FUNCTION_BLOCK FB_MY_SQL IMPLEMENTS I_DATABASE
VAR //General
	{attribute 'instance-path'} 
  {attribute 'noinit'} 
	strInstancePath:									                      STRING;
	bInit: 												                          BOOL:=TRUE;
	strFullObjectPath: 								                      STRING;
	stEvent:											                          ST_EVENT;
	bAck:												                            BOOL;
	
END_VAR
VAR   // From FB_init	
	itfLogEvents: 										                      I_HANDLE_EVENTS;
  itfOpMode:											                        I_OP_MODE; 
END_VAR                                      				
VAR	// Step chain control                				
  eSeq, eLastSeq, eNextSeq:					                      E_SEQ_DATABASE; 
                  				
  //eActiveSeqState, eLastActiveSeqState:                 E_SEQ_GENERAL;
	(*
  iInternalSeqStateCase, iLastInternalSeqStateCase:       INT:=0;       
	tonDelay, tonTimeOut, tonStepTime:						          TON;
	tDelay:													                        TIME := T#100MS;
	tTimeOut:												                        TIME := T#100MS;
	tTimeOutExt:											                      TIME := T#100MS;
	bDelayActive, bTimeOutActiveQuit, bTimeOutActiveNoQuit:	BOOL;//Timer Option
	bActiveStep, bDebugAcitve, bDebugNext:					        BOOL;//Debug Option
	i:														                          INT;
 	iError:													                        INT; //ERROR-CODE                    	                   		
	listLastSteps:											                    ARRAY[0..49] OF ST_LAST_STEPS;	
	strExtraInfo:											                      STRING; 
	eStep_Type:												                      E_STEP_STATE_TYPE; 
	bDebugModeActive:										                    BOOL;   
	bWaitForBreakpoint:										                  BOOL;
	bBreakpointActive:										                  BOOL;
	bDebugResume:											                      BOOL;   
	listBreakpoint:											                    ARRAY[0..10] OF  INT;    
*)
i:														                            INT;
stSeqCtrlGeneral:											                    ST_SEQ_CTRL_GEN;     	
END_VAR                                             		
VAR                                                 		
	bMethodeFromExtStarted:									                BOOL;
	bMethodeFromExtActive:									                BOOL;
	bMethodeFromExtDone:									                  BOOL;
	strTemp:												                        STRING;
END_VAR   
VAR
  fbSQLDatabase:            FB_SQLDatabaseEvt(sNetID := '', tTimeout := T#5S);
  fbSQLCommand:             FB_SQLCommandEvt(sNetID := '', tTimeout := T#5S);
  fbPLCDBCmd:               FB_PLCDBCmdEvt(sNetID := '', tTimeout := T#5S);
  fbPLCDBCreateEvt:         FB_PLCDBCreateEvt(sNetID := '', tTimeout := T#5S);
  fbPLCDBReadEvt:           FB_PLCDBReadEvt(sNetID:= '', tTimeout:= T#5S);
  fbPLCDBWriteEvt:          FB_PLCDBWriteEvt(sNetID := '', tTimeout := T#5S);
  udiDBID:                  UDINT;
  pDBID:                    POINTER TO UDINT;
  sCmd:                     STRING(5000);
  sTableName:               T_MaxString;
  sDBSymbolName:            STRING;
  pRecord:                  POINTER TO BYTE;
  cbRecord:                 UDINT;
  pValue:                   POINTER TO BYTE;
  cbValue:                  UDINT;
  pColumnNames:             POINTER TO ARRAY [0..MAX_DBCOLUMNS] OF STRING(50);
  cbColumnNames:            UDINT;
  pTableCfg:                POINTER TO ARRAY[0..MAX_DBCOLUMNS] OF ST_ColumnInfo;
  cbTableCfg:               UDINT;
  sOrderByColumn:           STRING(50);
  eOrderBy:                 E_OrderColumn;
  eOrderType:               E_OrderType;
  nStartIndex:              UDINT;
  nRecordCount:             UDINT;
  pData:                    POINTER TO BYTE;
  pData2:                   POINTER TO ST_StandardRecord;
  cbData:                   UDINT;
  pDatabaseConfig:          POINTER TO BYTE;
  cbDatabaseConfig:         UDINT;
  bCreateXMLConfig:         BOOL;
  sColumnNameToUpdate:      STRING;
  sColumnValToUpdate:       STRING;
  sColumnNameToSet:         STRING;
  sNewVal:                  STRING;
  eDBWriteMode:             E_WriteMode;
  nRingBuffParameter:       UDINT;
  stADSDevice:              ST_ADSDevice;
  stSymbol:                 ST_Symbol;
  pExpression:              POINTER TO BYTE;
  cbExpression:             UDINT;
  pParameter:               POINTER TO ARRAY[0..MAX_DBCOLUMNS] OF ST_ExpParameter;
  cbParameter:              UDINT; 
  pSQLCmd:                  POINTER TO BYTE;
  cbSQLCmd:                 UDINT;
  bResult:                  BOOL;
END_VAR                  	
VAR_TEMP                    	
	iTemp:										INT;
END_VAR

// Set FBs and Interfaces ready after switch internal step
IF stSeqCtrlGeneral.iInternalSeqStateCase <> stSeqCtrlGeneral.iLastInternalSeqStateCase AND NOT stSeqCtrlGeneral.bExitSetReadyState THEN
  IF TRUE
  THEN
    stSeqCtrlGeneral.bExitSetReadyState := TRUE;
  ELSE
    RETURN;
  END_IF
END_IF

stSeqCtrlGeneral.strObject := F_CreateObjectName(strInstancePath);

// First method call
_m_SequenceManager();
//_m_SaveLastStep();

CASE eSeq OF 
  E_SEQ_DATABASE.BASE:;
  
	E_SEQ_DATABASE.INIT: _m_Seq_INIT();
		IF TRUE
		AND (stSeqCtrlGeneral.eActiveSeqState = E_SEQ_GENERAL.DONE) 
		THEN
			eSeq := E_SEQ_DATABASE.BASE;
		END_IF
		
	E_SEQ_DATABASE.SETUP:;
  
	// Process
  E_SEQ_DATABASE.CREATE_DATABASE: _m_Seq_CREATE_DATABASE();
    IF TRUE
		AND (stSeqCtrlGeneral.eActiveSeqState = E_SEQ_GENERAL.DONE) 
		THEN
			eSeq := E_SEQ_DATABASE.BASE;
		END_IF
  
	E_SEQ_DATABASE.CONNECT:         _m_Seq_CONNECT();
    IF TRUE
		AND (stSeqCtrlGeneral.eActiveSeqState = E_SEQ_GENERAL.DONE) 
		THEN
			eSeq := E_SEQ_DATABASE.BASE;
		END_IF
    
  E_SEQ_DATABASE.EXECUTE_SIMPLIFY_CMD:  _m_Seq_EXECUTE_SIMPLIFY_CMD();
    IF TRUE
		AND (stSeqCtrlGeneral.eActiveSeqState = E_SEQ_GENERAL.DONE) 
		THEN
			eSeq := E_SEQ_DATABASE.BASE;
		END_IF
  
  E_SEQ_DATABASE.EXECUTE_CMD:     _m_Seq_EXECUTE_CMD();
    IF TRUE
		AND (stSeqCtrlGeneral.eActiveSeqState = E_SEQ_GENERAL.DONE) 
		THEN
			eSeq := E_SEQ_DATABASE.BASE;
		END_IF
    
  E_SEQ_DATABASE.TABLE_EXIST_CHECK:     _m_Seq_TABLE_EXIST_CHECK();
    IF TRUE
		AND (stSeqCtrlGeneral.eActiveSeqState = E_SEQ_GENERAL.DONE) 
		THEN
			eSeq := E_SEQ_DATABASE.BASE;
		END_IF
  
  E_SEQ_DATABASE.CREATE_TABLE:    _m_Seq_CREATE_TABLE();
    IF TRUE
		AND (stSeqCtrlGeneral.eActiveSeqState = E_SEQ_GENERAL.DONE) 
		THEN
			eSeq := E_SEQ_DATABASE.BASE;
		END_IF
  
  E_SEQ_DATABASE.WRITE:           _m_Seq_WRITE();
    IF TRUE
		AND (stSeqCtrlGeneral.eActiveSeqState = E_SEQ_GENERAL.DONE) 
		THEN
			eSeq := E_SEQ_DATABASE.BASE;
		END_IF
  
  E_SEQ_DATABASE.WRITE_STRUCT:    _m_Seq_WRITE_STRUCT();
    IF TRUE
		AND (stSeqCtrlGeneral.eActiveSeqState = E_SEQ_GENERAL.DONE) 
		THEN
			eSeq := E_SEQ_DATABASE.BASE;
		END_IF
  
  E_SEQ_DATABASE.WRITE_BY_SYMBOL: _m_Seq_WRITE_BY_SYMBOL();
    IF TRUE
		AND (stSeqCtrlGeneral.eActiveSeqState = E_SEQ_GENERAL.DONE) 
		THEN
			eSeq := E_SEQ_DATABASE.BASE;
		END_IF
  
  E_SEQ_DATABASE.OVERWRITE:       _m_Seq_OVERWRITE();
    IF TRUE
		AND (stSeqCtrlGeneral.eActiveSeqState = E_SEQ_GENERAL.DONE) 
		THEN
			eSeq := E_SEQ_DATABASE.BASE;
		END_IF
  
  E_SEQ_DATABASE.READ:            _m_Seq_READ();
    IF TRUE
		AND (stSeqCtrlGeneral.eActiveSeqState = E_SEQ_GENERAL.DONE) 
		THEN
			eSeq := E_SEQ_DATABASE.BASE;
		END_IF
  
  E_SEQ_DATABASE.READ_STRUCT:     _m_Seq_READ_STRUCT();
    IF TRUE
		AND (stSeqCtrlGeneral.eActiveSeqState = E_SEQ_GENERAL.DONE) 
		THEN
			eSeq := E_SEQ_DATABASE.BASE;
		END_IF
  
  E_SEQ_DATABASE.CLEAR_TABLE:     _m_Seq_CLEAR_TABLE();
    IF TRUE
		AND (stSeqCtrlGeneral.eActiveSeqState = E_SEQ_GENERAL.DONE) 
		THEN
			eSeq := E_SEQ_DATABASE.BASE;
		END_IF
  
  E_SEQ_DATABASE.DELETE_TABLE:    _m_Seq_DELETE_TABLE();
    IF TRUE
		AND (stSeqCtrlGeneral.eActiveSeqState = E_SEQ_GENERAL.DONE) 
		THEN
			eSeq := E_SEQ_DATABASE.BASE;
		END_IF
  
  E_SEQ_DATABASE.DISCONNECT:      _m_Seq_DISCONNECT();
    IF TRUE
		AND (stSeqCtrlGeneral.eActiveSeqState = E_SEQ_GENERAL.DONE) 
		THEN
			eSeq := E_SEQ_DATABASE.BASE;
		END_IF

  // End
	E_SEQ_DATABASE.END:;
	E_SEQ_DATABASE.ERROR_SEQ:;	
END_CASE

strTemp:=TO_STRING(eSeq);

METHOD PRIVATE _m_DebugManager
VAR_INPUT
	iStepID: int;
END_VAR
IF TRUE
AND THIS^.stSeqCtrlGeneral.bDebugModeActive 
AND NOT THIS^.stSeqCtrlGeneral.bActiveStep
THEN


THIS^.stSeqCtrlGeneral.bBreakpointActive:=FALSE;

FOR i:=0 TO 10 DO
	
	IF TRUE
	AND iStepID=THIS^.stSeqCtrlGeneral.listBreakpoint[i] 
	AND iStepID<>0
	THEN
		EXIT;
	END_IF
END_FOR
IF (i<=10) THEN
	THIS^.stSeqCtrlGeneral.bBreakpointActive:=TRUE;
END_IF

END_IF
END_METHOD

METHOD PRIVATE _m_Delay : BOOL
VAR_INPUT
	DelayTime:	TIME;
END_VAR
THIS^.stSeqCtrlGeneral.bDelayActive:=TRUE;
THIS^.stSeqCtrlGeneral.tDelay:=DelayTime;
_m_Delay:=FALSE;
IF THIS^.stSeqCtrlGeneral.tonDelay.Q THEN
	_m_Delay:=TRUE;
END_IF
END_METHOD

METHOD PRIVATE _m_GeneralStepSetting : BOOL
VAR_INPUT
	StepType:			    	E_STEP_STATE_TYPE;
	InfoTextID:					STRING(20);
	EnableDebug:	   			BOOL;	
	
END_VAR
IF THIS^.stSeqCtrlGeneral.bActiveStep THEN
	THIS^.stSeqCtrlGeneral.eStep_Type:=StepType;
	THIS^.stSeqCtrlGeneral.strExtraInfo:= GenLib.F_RET_TXTLIST_ENTRY(strPortNr:='851',strID:='',strTxtLstName:=InfoTextID);
END_IF
END_METHOD

METHOD PRIVATE _m_SaveLastStep : BOOL
VAR_INPUT
END_VAR
VAR
	i: dint;
END_VAR
IF NOT THIS^.stSeqCtrlGeneral.bActiveStep THEN
	
	FOR i:=49 TO 1 BY -1 DO
			stSeqCtrlGeneral.listLastSteps[i].strStepName:=stSeqCtrlGeneral.listLastSteps[i-1].strStepName;
			stSeqCtrlGeneral.listLastSteps[i].tStepTime:=stSeqCtrlGeneral.listLastSteps[i-1].tStepTime;
			stSeqCtrlGeneral.listLastSteps[i].tDelayTime:=stSeqCtrlGeneral.listLastSteps[i-1].tDelayTime;
	END_FOR
	stSeqCtrlGeneral.listLastSteps[0].strStepName:=TO_STRING(THIS^.eSeq);
	stSeqCtrlGeneral.listLastSteps[1].tStepTime:=THIS^.stSeqCtrlGeneral.tonStepTime.ET;
	stSeqCtrlGeneral.listLastSteps[1].tStepTime:=THIS^.stSeqCtrlGeneral.tonDelay.ET;
ELSE
	stSeqCtrlGeneral.listLastSteps[0].tStepTime:=THIS^.stSeqCtrlGeneral.tonStepTime.ET;
	stSeqCtrlGeneral.listLastSteps[0].tDelayTime:=THIS^.stSeqCtrlGeneral.tonDelay.ET;	
END_IF
END_METHOD

METHOD PRIVATE _m_Seq_CLEAR_TABLE : E_SEQ_PROCESS
VAR_INPUT
END_VAR
VAR
	ActiveSeq: STRING;
END_VAR
VAR
	
END_VAR
//THIS^._m_GeneralStepSetting(StepType:=E_STEP_STATE_TYPE.INIT,
ActiveSeq := TO_STRING(THIS^.eSeq);

CASE THIS^.stSeqCtrlGeneral.eActiveSeqState OF
E_SEQ_GENERAL.READY:;

	
E_SEQ_GENERAL.EXECUTE:;
	IF TRUE
	THEN
		THIS^.stSeqCtrlGeneral.eActiveSeqState := E_SEQ_GENERAL.RESET;
	END_IF
  
E_SEQ_GENERAL.RESET:;
	stSeqCtrlGeneral.iInternalSeqStateCase := 0;
	IF TRUE
	THEN
		THIS^.stSeqCtrlGeneral.eActiveSeqState := E_SEQ_GENERAL.BUSY;
	END_IF
  
E_SEQ_GENERAL.BUSY:;
	CASE THIS^.stSeqCtrlGeneral.iInternalSeqStateCase OF
    0:  // Connect to database
      IF TRUE 
      AND NOT THIS^.fbSQLDatabase.bConnected
			THEN 
        IF THIS^.fbSQLDatabase.Connect(THIS^.udiDBID) THEN
          IF THIS^.fbSQLDatabase.bError THEN
            THIS^.stSeqCtrlGeneral.eActiveSeqState := E_SEQ_GENERAL.ERROR;
          ELSE
            THIS^.stSeqCtrlGeneral.iInternalSeqStateCase := 10;
          END_IF
        END_IF
      ELSE
        THIS^.stSeqCtrlGeneral.iInternalSeqStateCase := 10;
			END_IF
      
		10:	// Create command
      IF TRUE 
			THEN 
        sCmd := 'DELETE FROM `';
        sCmd := CONCAT(sCmd, sTableName);
        sCmd := CONCAT(sCmd, '`');
        IF fbSQLDatabase.CreateCmd(ADR(fbSQLCommand)) THEN
          IF fbSqlDatabase.bError THEN
            THIS^.stSeqCtrlGeneral.eActiveSeqState := E_SEQ_GENERAL.ERROR;
          ELSE
            THIS^.stSeqCtrlGeneral.iInternalSeqStateCase := 20;  
          END_IF
        END_IF
			END_IF
      
		20: // Execute command
      IF TRUE 
			THEN
        IF fbSQLCommand.Execute(ADR(sCmd), SIZEOF(sCmd)) THEN
          IF fbSQLCommand.bError THEN
            THIS^.stSeqCtrlGeneral.eActiveSeqState := E_SEQ_GENERAL.ERROR;
          ELSE
            THIS^.stSeqCtrlGeneral.iInternalSeqStateCase := 30;
          END_IF
	      END_IF
			END_IF
      
    30:	// Disconnect
      IF TRUE 
			THEN 
        IF fbSQLDatabase.Disconnect() THEN
          IF fbSqlDatabase.bError THEN
            THIS^.stSeqCtrlGeneral.eActiveSeqState := E_SEQ_GENERAL.ERROR;
          ELSE
            THIS^.stSeqCtrlGeneral.iInternalSeqStateCase := 1000;
          END_IF
        END_IF
			END_IF
      
	ELSE
		THIS^.stSeqCtrlGeneral.eActiveSeqState := E_SEQ_GENERAL.DONE;  
	END_CASE
	THIS^.stSeqCtrlGeneral.strExtraInfo := CONCAT('Internal state: ', TO_STRING(THIS^.stSeqCtrlGeneral.iInternalSeqStateCase));

E_SEQ_GENERAL.DONE:;

E_SEQ_GENERAL.ERROR:;

E_SEQ_GENERAL.TIME_OUT:; 
IF TRUE
AND THIS^.stSeqCtrlGeneral.bTimeOutActiveQuit 
THEN
  THIS^.stSeqCtrlGeneral.strExtraInfo := 'Bitte quittieren und erneut testen';
  IF TRUE
  //AND itfOpMode.P_QUIT
  THEN
    THIS^.stSeqCtrlGeneral.eActiveSeqState := E_SEQ_GENERAL.EXECUTE;
	END_IF
  
END_IF

ELSE
  THIS^.stSeqCtrlGeneral.eActiveSeqState := E_SEQ_GENERAL.ERROR;
END_CASE
END_METHOD

METHOD PRIVATE _m_Seq_CONNECT : E_SEQ_PROCESS
VAR_INPUT
END_VAR
VAR
	ActiveSeq: STRING;
END_VAR
VAR
	
END_VAR
//THIS^._m_GeneralStepSetting(StepType:=E_STEP_STATE_TYPE.INIT,
ActiveSeq := TO_STRING(THIS^.eSeq);

CASE THIS^.stSeqCtrlGeneral.eActiveSeqState OF
E_SEQ_GENERAL.READY:;

	
E_SEQ_GENERAL.EXECUTE:;
	IF TRUE
	THEN
		THIS^.stSeqCtrlGeneral.eActiveSeqState := E_SEQ_GENERAL.RESET;
	END_IF
  
E_SEQ_GENERAL.RESET:;
	stSeqCtrlGeneral.iInternalSeqStateCase := 0;
	IF TRUE
	THEN
		THIS^.stSeqCtrlGeneral.eActiveSeqState := E_SEQ_GENERAL.BUSY;
	END_IF
  
E_SEQ_GENERAL.BUSY:;
	CASE THIS^.stSeqCtrlGeneral.iInternalSeqStateCase OF
		0:	// Entrance step --> Connect
      IF TRUE 
      AND NOT THIS^.fbSQLDatabase.bConnected
			THEN 
        IF THIS^.fbSQLDatabase.Connect(THIS^.udiDBID) THEN
          IF THIS^.fbSQLDatabase.bError THEN
            THIS^.stSeqCtrlGeneral.eActiveSeqState := E_SEQ_GENERAL.ERROR;
          ELSE
            THIS^.stSeqCtrlGeneral.iInternalSeqStateCase := 1000;
          END_IF
        END_IF
      ELSE
        THIS^.stSeqCtrlGeneral.iInternalSeqStateCase := 1000;
			END_IF
      
	ELSE
		THIS^.stSeqCtrlGeneral.eActiveSeqState := E_SEQ_GENERAL.DONE;  
	END_CASE
	THIS^.stSeqCtrlGeneral.strExtraInfo := CONCAT('Internal state: ', TO_STRING(THIS^.stSeqCtrlGeneral.iInternalSeqStateCase));

E_SEQ_GENERAL.DONE:;

E_SEQ_GENERAL.ERROR:;

E_SEQ_GENERAL.TIME_OUT:; 
IF TRUE
AND THIS^.stSeqCtrlGeneral.bTimeOutActiveQuit 
THEN
  THIS^.stSeqCtrlGeneral.strExtraInfo := 'Bitte quittieren und erneut testen';
  IF TRUE
  //AND itfOpMode.P_QUIT
  THEN
    THIS^.stSeqCtrlGeneral.eActiveSeqState := E_SEQ_GENERAL.EXECUTE;
	END_IF
  
END_IF

ELSE
  THIS^.stSeqCtrlGeneral.eActiveSeqState := E_SEQ_GENERAL.ERROR;
END_CASE
END_METHOD

METHOD PRIVATE _m_Seq_CREATE_DATABASE : E_SEQ_PROCESS
VAR_INPUT
END_VAR
VAR
	ActiveSeq: STRING;
END_VAR
VAR
  stTemp:                     STRING;
END_VAR
//THIS^._m_GeneralStepSetting(StepType:=E_STEP_STATE_TYPE.INIT,
ActiveSeq := TO_STRING(THIS^.eSeq);

CASE THIS^.stSeqCtrlGeneral.eActiveSeqState OF
E_SEQ_GENERAL.READY:;

	
E_SEQ_GENERAL.EXECUTE:;
	IF TRUE
	THEN
		THIS^.stSeqCtrlGeneral.eActiveSeqState := E_SEQ_GENERAL.RESET;
	END_IF
  
E_SEQ_GENERAL.RESET:;
	stSeqCtrlGeneral.iInternalSeqStateCase := 0;
	IF TRUE
	THEN
		THIS^.stSeqCtrlGeneral.eActiveSeqState := E_SEQ_GENERAL.BUSY;
	END_IF
  
E_SEQ_GENERAL.BUSY:;
	CASE THIS^.stSeqCtrlGeneral.iInternalSeqStateCase OF
    0:	// Create database
      IF TRUE 
			THEN
        IF fbPLCDBCreateEvt.Database(
          pDatabaseConfig:= pDatabaseConfig,
          cbDatabaseConfig:= cbDatabaseConfig,
          bCreateXMLConfig:= bCreateXMLConfig,
          pDBID := pDBID)
        THEN
          IF fbPLCDBCreateEvt.bError THEN
            THIS^.stSeqCtrlGeneral.eActiveSeqState := E_SEQ_GENERAL.ERROR; 
          ELSE
            THIS^.stSeqCtrlGeneral.iInternalSeqStateCase := 1000;
          END_IF
        END_IF
      END_IF
      
	ELSE
		THIS^.stSeqCtrlGeneral.eActiveSeqState := E_SEQ_GENERAL.DONE;  
	END_CASE
	THIS^.stSeqCtrlGeneral.strExtraInfo := CONCAT('Internal state: ', TO_STRING(THIS^.stSeqCtrlGeneral.iInternalSeqStateCase));

E_SEQ_GENERAL.DONE:;

E_SEQ_GENERAL.ERROR:;

E_SEQ_GENERAL.TIME_OUT:; 
IF TRUE
AND THIS^.stSeqCtrlGeneral.bTimeOutActiveQuit 
THEN
  THIS^.stSeqCtrlGeneral.strExtraInfo := 'Bitte quittieren und erneut testen';
  IF TRUE
  //AND itfOpMode.P_QUIT
  THEN
    THIS^.stSeqCtrlGeneral.eActiveSeqState := E_SEQ_GENERAL.EXECUTE;
	END_IF
  
END_IF

ELSE
  THIS^.stSeqCtrlGeneral.eActiveSeqState := E_SEQ_GENERAL.ERROR;
END_CASE
END_METHOD

METHOD PRIVATE _m_Seq_CREATE_TABLE : E_SEQ_PROCESS
VAR_INPUT
END_VAR
VAR
	ActiveSeq: STRING;
END_VAR
VAR
  stTemp:                     STRING;
END_VAR
//THIS^._m_GeneralStepSetting(StepType:=E_STEP_STATE_TYPE.INIT,
ActiveSeq := TO_STRING(THIS^.eSeq);

CASE THIS^.stSeqCtrlGeneral.eActiveSeqState OF
E_SEQ_GENERAL.READY:;

	
E_SEQ_GENERAL.EXECUTE:;
	IF TRUE
	THEN
		THIS^.stSeqCtrlGeneral.eActiveSeqState := E_SEQ_GENERAL.RESET;
	END_IF
  
E_SEQ_GENERAL.RESET:;
	stSeqCtrlGeneral.iInternalSeqStateCase := 0;
	IF TRUE
	THEN
		THIS^.stSeqCtrlGeneral.eActiveSeqState := E_SEQ_GENERAL.BUSY;
	END_IF
  
E_SEQ_GENERAL.BUSY:;
	CASE THIS^.stSeqCtrlGeneral.iInternalSeqStateCase OF
    0:	// Create table
      IF TRUE 
			THEN
        IF fbPLCDBCreateEvt.Table(hDBID:= udiDBID,
                                  sTableName:= sTableName, 
                                  pTableCfg:= THIS^.pTableCfg, 
                                  cbTableCfg:= THIS^.cbTableCfg)
        THEN
          IF fbPLCDBCreateEvt.bError THEN
            THIS^.stSeqCtrlGeneral.eActiveSeqState := E_SEQ_GENERAL.ERROR; 
          ELSE
            THIS^.stSeqCtrlGeneral.iInternalSeqStateCase := 1000;
          END_IF
        END_IF
      END_IF
      
	ELSE
		THIS^.stSeqCtrlGeneral.eActiveSeqState := E_SEQ_GENERAL.DONE;  
	END_CASE
	THIS^.stSeqCtrlGeneral.strExtraInfo := CONCAT('Internal state: ', TO_STRING(THIS^.stSeqCtrlGeneral.iInternalSeqStateCase));

E_SEQ_GENERAL.DONE:;

E_SEQ_GENERAL.ERROR:;

E_SEQ_GENERAL.TIME_OUT:; 
IF TRUE
AND THIS^.stSeqCtrlGeneral.bTimeOutActiveQuit 
THEN
  THIS^.stSeqCtrlGeneral.strExtraInfo := 'Bitte quittieren und erneut testen';
  IF TRUE
  //AND itfOpMode.P_QUIT
  THEN
    THIS^.stSeqCtrlGeneral.eActiveSeqState := E_SEQ_GENERAL.EXECUTE;
	END_IF
  
END_IF

ELSE
  THIS^.stSeqCtrlGeneral.eActiveSeqState := E_SEQ_GENERAL.ERROR;
END_CASE
END_METHOD

METHOD PRIVATE _m_Seq_DELETE_TABLE : E_SEQ_PROCESS
VAR_INPUT
END_VAR
VAR
	ActiveSeq: STRING;
END_VAR
VAR
	
END_VAR
//THIS^._m_GeneralStepSetting(StepType:=E_STEP_STATE_TYPE.INIT,
ActiveSeq := TO_STRING(THIS^.eSeq);

CASE THIS^.stSeqCtrlGeneral.eActiveSeqState OF
E_SEQ_GENERAL.READY:;

	
E_SEQ_GENERAL.EXECUTE:;
	IF TRUE
	THEN
		THIS^.stSeqCtrlGeneral.eActiveSeqState := E_SEQ_GENERAL.RESET;
	END_IF
  
E_SEQ_GENERAL.RESET:;
	stSeqCtrlGeneral.iInternalSeqStateCase := 0;
	IF TRUE
	THEN
		THIS^.stSeqCtrlGeneral.eActiveSeqState := E_SEQ_GENERAL.BUSY;
	END_IF
  
E_SEQ_GENERAL.BUSY:;
	CASE THIS^.stSeqCtrlGeneral.iInternalSeqStateCase OF
    0:  // Connect to database
      IF TRUE 
      AND NOT THIS^.fbSQLDatabase.bConnected
			THEN 
        IF THIS^.fbSQLDatabase.Connect(THIS^.udiDBID) THEN
          IF THIS^.fbSQLDatabase.bError THEN
            THIS^.stSeqCtrlGeneral.eActiveSeqState := E_SEQ_GENERAL.ERROR;
          ELSE
            THIS^.stSeqCtrlGeneral.iInternalSeqStateCase := 10;
          END_IF
        END_IF
      ELSE
        THIS^.stSeqCtrlGeneral.iInternalSeqStateCase := 10;
			END_IF
      
		10:	// Create command
      IF TRUE 
			THEN 
        sCmd := 'DROP TABLE `';
        sCmd := CONCAT(sCmd, sTableName);
        sCmd := CONCAT(sCmd, '`');
        IF fbSQLDatabase.CreateCmd(ADR(fbSQLCommand)) THEN
          IF fbSqlDatabase.bError THEN
            THIS^.stSeqCtrlGeneral.eActiveSeqState := E_SEQ_GENERAL.ERROR;
          ELSE
            THIS^.stSeqCtrlGeneral.iInternalSeqStateCase := 20;  
          END_IF
        END_IF
			END_IF
      
		20: // Execute command
      IF TRUE 
			THEN
        IF fbSQLCommand.Execute(ADR(sCmd), SIZEOF(sCmd)) THEN
          IF fbSQLCommand.bError THEN
            THIS^.stSeqCtrlGeneral.eActiveSeqState := E_SEQ_GENERAL.ERROR;
          ELSE
            THIS^.stSeqCtrlGeneral.iInternalSeqStateCase := 30;
          END_IF
	      END_IF
			END_IF
      
    30:	// Disconnect
      IF TRUE 
			THEN 
        IF fbSQLDatabase.Disconnect() THEN
          IF fbSqlDatabase.bError THEN
            THIS^.stSeqCtrlGeneral.eActiveSeqState := E_SEQ_GENERAL.ERROR;
          ELSE
            THIS^.stSeqCtrlGeneral.iInternalSeqStateCase := 1000;
          END_IF
        END_IF
			END_IF
      
	ELSE
		THIS^.stSeqCtrlGeneral.eActiveSeqState := E_SEQ_GENERAL.DONE;  
	END_CASE
	THIS^.stSeqCtrlGeneral.strExtraInfo := CONCAT('Internal state: ', TO_STRING(THIS^.stSeqCtrlGeneral.iInternalSeqStateCase));

E_SEQ_GENERAL.DONE:;

E_SEQ_GENERAL.ERROR:;

E_SEQ_GENERAL.TIME_OUT:; 
IF TRUE
AND THIS^.stSeqCtrlGeneral.bTimeOutActiveQuit 
THEN
  THIS^.stSeqCtrlGeneral.strExtraInfo := 'Bitte quittieren und erneut testen';
  IF TRUE
  //AND itfOpMode.P_QUIT
  THEN
    THIS^.stSeqCtrlGeneral.eActiveSeqState := E_SEQ_GENERAL.EXECUTE;
	END_IF
  
END_IF

ELSE
  THIS^.stSeqCtrlGeneral.eActiveSeqState := E_SEQ_GENERAL.ERROR;
END_CASE
END_METHOD

METHOD PRIVATE _m_Seq_DISCONNECT : E_SEQ_PROCESS
VAR_INPUT
END_VAR
VAR
	ActiveSeq: STRING;
END_VAR
VAR
	
END_VAR
//THIS^._m_GeneralStepSetting(StepType:=E_STEP_STATE_TYPE.INIT,
ActiveSeq := TO_STRING(THIS^.eSeq);

CASE THIS^.stSeqCtrlGeneral.eActiveSeqState OF
E_SEQ_GENERAL.READY:;

	
E_SEQ_GENERAL.EXECUTE:;
	IF TRUE
	THEN
		THIS^.stSeqCtrlGeneral.eActiveSeqState := E_SEQ_GENERAL.RESET;
	END_IF
  
E_SEQ_GENERAL.RESET:;
	stSeqCtrlGeneral.iInternalSeqStateCase := 0;
	IF TRUE
	THEN
		THIS^.stSeqCtrlGeneral.eActiveSeqState := E_SEQ_GENERAL.BUSY;
	END_IF
  
E_SEQ_GENERAL.BUSY:;
	CASE THIS^.stSeqCtrlGeneral.iInternalSeqStateCase OF
		0:	// Entrance step --> Disconnect
      IF TRUE 
			THEN 
        IF fbSQLDatabase.Disconnect() THEN
          IF fbSqlDatabase.bError THEN
            THIS^.stSeqCtrlGeneral.eActiveSeqState := E_SEQ_GENERAL.ERROR;
          ELSE
            THIS^.stSeqCtrlGeneral.iInternalSeqStateCase := 1000;
          END_IF
        END_IF
			END_IF
      
	ELSE
		THIS^.stSeqCtrlGeneral.eActiveSeqState := E_SEQ_GENERAL.DONE;  
	END_CASE
	THIS^.stSeqCtrlGeneral.strExtraInfo := CONCAT('Internal state: ', TO_STRING(THIS^.stSeqCtrlGeneral.iInternalSeqStateCase));

E_SEQ_GENERAL.DONE:;

E_SEQ_GENERAL.ERROR:;

E_SEQ_GENERAL.TIME_OUT:; 
IF TRUE
AND THIS^.stSeqCtrlGeneral.bTimeOutActiveQuit 
THEN
  THIS^.stSeqCtrlGeneral.strExtraInfo := 'Bitte quittieren und erneut testen';
  IF TRUE
  //AND itfOpMode.P_QUIT
  THEN
    THIS^.stSeqCtrlGeneral.eActiveSeqState := E_SEQ_GENERAL.EXECUTE;
	END_IF
  
END_IF

ELSE
  THIS^.stSeqCtrlGeneral.eActiveSeqState := E_SEQ_GENERAL.ERROR;
END_CASE
END_METHOD

METHOD PRIVATE _m_Seq_EXECUTE_CMD : E_SEQ_PROCESS
VAR_INPUT
END_VAR
VAR
	ActiveSeq: STRING;
END_VAR
//THIS^._m_GeneralStepSetting(StepType:=E_STEP_STATE_TYPE.INIT,
ActiveSeq := TO_STRING(THIS^.eSeq);

CASE THIS^.stSeqCtrlGeneral.eActiveSeqState OF
E_SEQ_GENERAL.READY:;

	
E_SEQ_GENERAL.EXECUTE:;
	IF TRUE
	THEN
		THIS^.stSeqCtrlGeneral.eActiveSeqState := E_SEQ_GENERAL.RESET;
	END_IF
  
E_SEQ_GENERAL.RESET:;
	stSeqCtrlGeneral.iInternalSeqStateCase := 0;
	IF TRUE
	THEN
		THIS^.stSeqCtrlGeneral.eActiveSeqState := E_SEQ_GENERAL.BUSY;
	END_IF
  
E_SEQ_GENERAL.BUSY:;
	CASE THIS^.stSeqCtrlGeneral.iInternalSeqStateCase OF
    0:	// Execute command
      IF TRUE 
			THEN 
        IF fbPLCDBCmd.Execute(hDBID:= THIS^.udiDBID, 
                              pExpression:= pExpression, 
                              cbExpression:= cbExpression, 
                              pData:= pData, 
                              cbData:= cbData, 
                              pParameter:= pParameter, 
                              cbParameter:= cbParameter) 
        THEN
          IF fbPLCDBWriteEvt.bError THEN
            THIS^.stSeqCtrlGeneral.eActiveSeqState := E_SEQ_GENERAL.ERROR; 
          ELSE
            THIS^.stSeqCtrlGeneral.iInternalSeqStateCase := 1000;
          END_IF
        END_IF
			END_IF
      
	ELSE
		THIS^.stSeqCtrlGeneral.eActiveSeqState := E_SEQ_GENERAL.DONE;  
	END_CASE
	THIS^.stSeqCtrlGeneral.strExtraInfo := CONCAT('Internal state: ', TO_STRING(THIS^.stSeqCtrlGeneral.iInternalSeqStateCase));

E_SEQ_GENERAL.DONE:;

E_SEQ_GENERAL.ERROR:;

E_SEQ_GENERAL.TIME_OUT:; 
IF TRUE
AND THIS^.stSeqCtrlGeneral.bTimeOutActiveQuit 
THEN
  THIS^.stSeqCtrlGeneral.strExtraInfo := 'Bitte quittieren und erneut testen';
  IF TRUE
  //AND itfOpMode.P_QUIT
  THEN
    THIS^.stSeqCtrlGeneral.eActiveSeqState := E_SEQ_GENERAL.EXECUTE;
	END_IF
  
END_IF

ELSE
  THIS^.stSeqCtrlGeneral.eActiveSeqState := E_SEQ_GENERAL.ERROR;
END_CASE
END_METHOD

METHOD PRIVATE _m_Seq_EXECUTE_SIMPLIFY_CMD : E_SEQ_PROCESS
VAR_INPUT
END_VAR
VAR
	ActiveSeq: STRING;
END_VAR
//THIS^._m_GeneralStepSetting(StepType:=E_STEP_STATE_TYPE.INIT,
ActiveSeq := TO_STRING(THIS^.eSeq);

CASE THIS^.stSeqCtrlGeneral.eActiveSeqState OF
E_SEQ_GENERAL.READY:;

	
E_SEQ_GENERAL.EXECUTE:;
	IF TRUE
	THEN
		THIS^.stSeqCtrlGeneral.eActiveSeqState := E_SEQ_GENERAL.RESET;
	END_IF
  
E_SEQ_GENERAL.RESET:;
	stSeqCtrlGeneral.iInternalSeqStateCase := 0;
	IF TRUE
	THEN
		THIS^.stSeqCtrlGeneral.eActiveSeqState := E_SEQ_GENERAL.BUSY;
	END_IF
  
E_SEQ_GENERAL.BUSY:;
	CASE THIS^.stSeqCtrlGeneral.iInternalSeqStateCase OF
    0:  // Connect to database
      IF TRUE 
      AND NOT THIS^.fbSQLDatabase.bConnected
			THEN 
        IF THIS^.fbSQLDatabase.Connect(THIS^.udiDBID) THEN
          IF THIS^.fbSQLDatabase.bError THEN
            THIS^.stSeqCtrlGeneral.eActiveSeqState := E_SEQ_GENERAL.ERROR;
          ELSE
            THIS^.stSeqCtrlGeneral.iInternalSeqStateCase := 10;
          END_IF
        END_IF
      ELSE
        THIS^.stSeqCtrlGeneral.iInternalSeqStateCase := 10;
			END_IF

    10:	// Execute command
      IF TRUE 
			THEN 
        IF fbSQLCommand.Execute(THIS^.pSQLCmd, THIS^.cbSQLCmd) THEN
          IF fbPLCDBWriteEvt.bError THEN
            THIS^.stSeqCtrlGeneral.eActiveSeqState := E_SEQ_GENERAL.ERROR; 
          ELSE
            THIS^.stSeqCtrlGeneral.iInternalSeqStateCase := 20;
          END_IF
        END_IF
			END_IF
      
    20:	// Disconnect
      IF TRUE 
			THEN 
        IF fbSQLDatabase.Disconnect() THEN
          IF fbSqlDatabase.bError THEN
            THIS^.stSeqCtrlGeneral.eActiveSeqState := E_SEQ_GENERAL.ERROR;
          ELSE
            THIS^.stSeqCtrlGeneral.iInternalSeqStateCase := 1000;
          END_IF
        END_IF
			END_IF
      
	ELSE
		THIS^.stSeqCtrlGeneral.eActiveSeqState := E_SEQ_GENERAL.DONE;  
	END_CASE
	THIS^.stSeqCtrlGeneral.strExtraInfo := CONCAT('Internal state: ', TO_STRING(THIS^.stSeqCtrlGeneral.iInternalSeqStateCase));

E_SEQ_GENERAL.DONE:;

E_SEQ_GENERAL.ERROR:;

E_SEQ_GENERAL.TIME_OUT:; 
IF TRUE
AND THIS^.stSeqCtrlGeneral.bTimeOutActiveQuit 
THEN
  THIS^.stSeqCtrlGeneral.strExtraInfo := 'Bitte quittieren und erneut testen';
  IF TRUE
  //AND itfOpMode.P_QUIT
  THEN
    THIS^.stSeqCtrlGeneral.eActiveSeqState := E_SEQ_GENERAL.EXECUTE;
	END_IF
  
END_IF

ELSE
  THIS^.stSeqCtrlGeneral.eActiveSeqState := E_SEQ_GENERAL.ERROR;
END_CASE
END_METHOD

METHOD PRIVATE _m_Seq_INIT : E_SEQ_PROCESS
VAR_INPUT
END_VAR
VAR
	ActiveSeq: STRING;
END_VAR
VAR
	
END_VAR
//THIS^._m_GeneralStepSetting(StepType:=E_STEP_STATE_TYPE.INIT,
ActiveSeq := TO_STRING(THIS^.eSeq);

CASE THIS^.stSeqCtrlGeneral.eActiveSeqState OF
E_SEQ_GENERAL.READY:;

	
E_SEQ_GENERAL.EXECUTE:;
	IF TRUE
	THEN
		THIS^.stSeqCtrlGeneral.eActiveSeqState := E_SEQ_GENERAL.RESET;
	END_IF
E_SEQ_GENERAL.RESET:;
	stSeqCtrlGeneral.iInternalSeqStateCase := 0;
  
	IF TRUE
	THEN
		THIS^.stSeqCtrlGeneral.eActiveSeqState := E_SEQ_GENERAL.BUSY;
	END_IF
E_SEQ_GENERAL.BUSY:;
	CASE THIS^.stSeqCtrlGeneral.iInternalSeqStateCase OF
		0:	// Entrance step
      IF TRUE
			THEN 
				IF fbSQLDatabase.Disconnect() THEN
          IF fbSqlDatabase.bError THEN
            THIS^.stSeqCtrlGeneral.eActiveSeqState := E_SEQ_GENERAL.ERROR;
          ELSE
            THIS^.stSeqCtrlGeneral.iInternalSeqStateCase := 1000;
          END_IF
        END_IF
			END_IF
      
	ELSE
		THIS^.stSeqCtrlGeneral.eActiveSeqState := E_SEQ_GENERAL.DONE;  
	END_CASE
	THIS^.stSeqCtrlGeneral.strExtraInfo := CONCAT('Internal state: ', TO_STRING(THIS^.stSeqCtrlGeneral.iInternalSeqStateCase));
E_SEQ_GENERAL.DONE:;
E_SEQ_GENERAL.ERROR:;
E_SEQ_GENERAL.TIME_OUT:; 

IF TRUE
AND THIS^.stSeqCtrlGeneral.bTimeOutActiveQuit 
THEN
  THIS^.stSeqCtrlGeneral.strExtraInfo := 'Bitte quittieren und erneut testen';
  IF TRUE
  //AND itfOpMode.P_QUIT
  THEN
    THIS^.stSeqCtrlGeneral.eActiveSeqState := E_SEQ_GENERAL.EXECUTE;
	END_IF
  
END_IF

ELSE
  THIS^.stSeqCtrlGeneral.eActiveSeqState := E_SEQ_GENERAL.ERROR;
END_CASE
END_METHOD

METHOD PRIVATE _m_Seq_OVERWRITE : E_SEQ_PROCESS
VAR_INPUT
END_VAR
VAR
	ActiveSeq: STRING;
END_VAR
VAR
	sTableName:                 STRING;
  sColumnNameToUpdate:        STRING;
  sColumnValToUpdate:         STRING;
  sColumnNameToSet:           STRING;
  sNewVal:                    STRING;
END_VAR
//THIS^._m_GeneralStepSetting(StepType:=E_STEP_STATE_TYPE.INIT,
ActiveSeq := TO_STRING(THIS^.eSeq);

CASE THIS^.stSeqCtrlGeneral.eActiveSeqState OF
E_SEQ_GENERAL.READY:;

	
E_SEQ_GENERAL.EXECUTE:;
	IF TRUE
	THEN
		THIS^.stSeqCtrlGeneral.eActiveSeqState := E_SEQ_GENERAL.RESET;
	END_IF
  
E_SEQ_GENERAL.RESET:;
	stSeqCtrlGeneral.iInternalSeqStateCase := 0;
	IF TRUE
	THEN
		THIS^.stSeqCtrlGeneral.eActiveSeqState := E_SEQ_GENERAL.BUSY;
	END_IF
  
E_SEQ_GENERAL.BUSY:;
	CASE THIS^.stSeqCtrlGeneral.iInternalSeqStateCase OF
		0:  // Connect to database
      IF TRUE 
      AND NOT THIS^.fbSQLDatabase.bConnected
			THEN 
        IF THIS^.fbSQLDatabase.Connect(THIS^.udiDBID) THEN
          IF THIS^.fbSQLDatabase.bError THEN
            THIS^.stSeqCtrlGeneral.eActiveSeqState := E_SEQ_GENERAL.ERROR;
          ELSE
            THIS^.stSeqCtrlGeneral.iInternalSeqStateCase := 10;
          END_IF
        END_IF
      ELSE
        THIS^.stSeqCtrlGeneral.iInternalSeqStateCase := 10;
			END_IF

    10:	// Create command
      IF TRUE 
			THEN 
        sCmd := 'SET SQL_SAFE_UPDATES = 0; UPDATE `';
        sCmd := CONCAT(sCmd, THIS^.sTableName);
        sCmd := CONCAT(sCmd, '` SET ');
        sCmd := CONCAT(sCmd, THIS^.sColumnNameToSet);
        sCmd := CONCAT(sCmd, ' = $'');
        sCmd := CONCAT(sCmd, THIS^.sNewVal);
        sCmd := CONCAT(sCmd, '$' WHERE ');
        sCmd := CONCAT(sCmd, THIS^.sColumnNameToUpdate);
        sCmd := CONCAT(sCmd, ' = $'');
        sCmd := CONCAT(sCmd, THIS^.sColumnValToUpdate);
        sCmd := CONCAT(sCmd, '$';');
        IF fbSQLDatabase.CreateCmd(ADR(fbSQLCommand)) THEN
          IF fbSqlDatabase.bError THEN
            THIS^.stSeqCtrlGeneral.eActiveSeqState := E_SEQ_GENERAL.ERROR;
          ELSE
            THIS^.stSeqCtrlGeneral.iInternalSeqStateCase := 20;  
          END_IF
        END_IF
			END_IF
      
		20: // Execute command
      IF TRUE 
			THEN
        IF fbSQLCommand.Execute(ADR(sCmd), SIZEOF(sCmd)) THEN
          IF fbSQLCommand.bError THEN
            THIS^.stSeqCtrlGeneral.eActiveSeqState := E_SEQ_GENERAL.ERROR;
          ELSE
            THIS^.stSeqCtrlGeneral.iInternalSeqStateCase := 30;
          END_IF
	      END_IF
			END_IF
      
    30:	// Disconnect
      IF TRUE 
			THEN 
        IF fbSQLDatabase.Disconnect() THEN
          IF fbSqlDatabase.bError THEN
            THIS^.stSeqCtrlGeneral.eActiveSeqState := E_SEQ_GENERAL.ERROR;
          ELSE
            THIS^.stSeqCtrlGeneral.iInternalSeqStateCase := 1000;
          END_IF
        END_IF
			END_IF
      
	ELSE
		THIS^.stSeqCtrlGeneral.eActiveSeqState := E_SEQ_GENERAL.DONE;  
	END_CASE
	THIS^.stSeqCtrlGeneral.strExtraInfo := CONCAT('Internal state: ', TO_STRING(THIS^.stSeqCtrlGeneral.iInternalSeqStateCase));

E_SEQ_GENERAL.DONE:;

E_SEQ_GENERAL.ERROR:;

E_SEQ_GENERAL.TIME_OUT:; 
IF TRUE
AND THIS^.stSeqCtrlGeneral.bTimeOutActiveQuit 
THEN
  THIS^.stSeqCtrlGeneral.strExtraInfo := 'Bitte quittieren und erneut testen';
  IF TRUE
  //AND itfOpMode.P_QUIT
  THEN
    THIS^.stSeqCtrlGeneral.eActiveSeqState := E_SEQ_GENERAL.EXECUTE;
	END_IF
  
END_IF

ELSE
  THIS^.stSeqCtrlGeneral.eActiveSeqState := E_SEQ_GENERAL.ERROR;
END_CASE
END_METHOD

METHOD PRIVATE _m_Seq_READ : E_SEQ_PROCESS
VAR_INPUT
END_VAR
VAR
	ActiveSeq: STRING;
END_VAR
VAR
	
END_VAR
//THIS^._m_GeneralStepSetting(StepType:=E_STEP_STATE_TYPE.INIT,
ActiveSeq := TO_STRING(THIS^.eSeq);

CASE THIS^.stSeqCtrlGeneral.eActiveSeqState OF
E_SEQ_GENERAL.READY:;

	
E_SEQ_GENERAL.EXECUTE:;
	IF TRUE
	THEN
		THIS^.stSeqCtrlGeneral.eActiveSeqState := E_SEQ_GENERAL.RESET;
	END_IF
  
E_SEQ_GENERAL.RESET:;
	stSeqCtrlGeneral.iInternalSeqStateCase := 0;
	IF TRUE
	THEN
		THIS^.stSeqCtrlGeneral.eActiveSeqState := E_SEQ_GENERAL.BUSY;
	END_IF
  
E_SEQ_GENERAL.BUSY:;
	CASE THIS^.stSeqCtrlGeneral.iInternalSeqStateCase OF
		0:	// Entrance step --> Read struct
      IF TRUE 
			THEN 
        IF fbPLCDBReadEvt.Read(
          hDBID:= THIS^.udiDBID, 
          sTableName:= THIS^.sTableName, 
          sDBSymbolName:= THIS^.sDBSymbolName, 
          eOrderBy:= THIS^.eOrderBy, 
          eOrderType:= THIS^.eOrderType, 
          nStartIndex:= THIS^.nStartIndex, 
          nRecordCount:= THIS^.nRecordCount, 
          pData:= THIS^.pData2, 
          cbData:= THIS^.cbData)
        THEN
          IF fbPLCDBReadEvt.bError THEN
            THIS^.stSeqCtrlGeneral.eActiveSeqState := E_SEQ_GENERAL.ERROR;
          ELSE
            THIS^.stSeqCtrlGeneral.iInternalSeqStateCase := 1000;
          END_IF
        END_IF
			END_IF
      
	ELSE
		THIS^.stSeqCtrlGeneral.eActiveSeqState := E_SEQ_GENERAL.DONE;  
	END_CASE
	THIS^.stSeqCtrlGeneral.strExtraInfo := CONCAT('Internal state: ', TO_STRING(THIS^.stSeqCtrlGeneral.iInternalSeqStateCase));

E_SEQ_GENERAL.DONE:;

E_SEQ_GENERAL.ERROR:;

E_SEQ_GENERAL.TIME_OUT:; 
IF TRUE
AND THIS^.stSeqCtrlGeneral.bTimeOutActiveQuit 
THEN
  THIS^.stSeqCtrlGeneral.strExtraInfo := 'Bitte quittieren und erneut testen';
  IF TRUE
  //AND itfOpMode.P_QUIT
  THEN
    THIS^.stSeqCtrlGeneral.eActiveSeqState := E_SEQ_GENERAL.EXECUTE;
	END_IF
  
END_IF

ELSE
  THIS^.stSeqCtrlGeneral.eActiveSeqState := E_SEQ_GENERAL.ERROR;
END_CASE
END_METHOD

METHOD PRIVATE _m_Seq_READ_STRUCT : E_SEQ_PROCESS
VAR_INPUT
END_VAR
VAR
	ActiveSeq: STRING;
END_VAR
VAR
	
END_VAR
//THIS^._m_GeneralStepSetting(StepType:=E_STEP_STATE_TYPE.INIT,
ActiveSeq := TO_STRING(THIS^.eSeq);

CASE THIS^.stSeqCtrlGeneral.eActiveSeqState OF
E_SEQ_GENERAL.READY:;

	
E_SEQ_GENERAL.EXECUTE:;
	IF TRUE
	THEN
		THIS^.stSeqCtrlGeneral.eActiveSeqState := E_SEQ_GENERAL.RESET;
	END_IF
  
E_SEQ_GENERAL.RESET:;
	stSeqCtrlGeneral.iInternalSeqStateCase := 0;
	IF TRUE
	THEN
		THIS^.stSeqCtrlGeneral.eActiveSeqState := E_SEQ_GENERAL.BUSY;
	END_IF
  
E_SEQ_GENERAL.BUSY:;
	CASE THIS^.stSeqCtrlGeneral.iInternalSeqStateCase OF
		0:	// Entrance step --> Read struct
      IF TRUE 
			THEN 
        IF fbPLCDBReadEvt.ReadStruct(hDBID:= THIS^.udiDBID, 
                                     sTableName:= THIS^.sTableName, 
                                     pColumnNames:= THIS^.pColumnNames,
                                     cbColumnNames:= THIS^.cbColumnNames,
                                     sOrderByColumn:= THIS^.sOrderByColumn,
                                     eOrderType:= THIS^.eOrderType, 
                                     nStartIndex:= THIS^.nStartIndex, 
                                     nRecordCount:= THIS^.nRecordCount, 
                                     pData:= THIS^.pData, 
                                     cbData:= THIS^.cbData) 
        THEN
          IF fbPLCDBReadEvt.bError THEN
            THIS^.stSeqCtrlGeneral.eActiveSeqState := E_SEQ_GENERAL.ERROR;
          ELSE
            THIS^.stSeqCtrlGeneral.iInternalSeqStateCase := 1000;
          END_IF
        END_IF
			END_IF
      
	ELSE
		THIS^.stSeqCtrlGeneral.eActiveSeqState := E_SEQ_GENERAL.DONE;  
	END_CASE
	THIS^.stSeqCtrlGeneral.strExtraInfo := CONCAT('Internal state: ', TO_STRING(THIS^.stSeqCtrlGeneral.iInternalSeqStateCase));

E_SEQ_GENERAL.DONE:;

E_SEQ_GENERAL.ERROR:;

E_SEQ_GENERAL.TIME_OUT:; 
IF TRUE
AND THIS^.stSeqCtrlGeneral.bTimeOutActiveQuit 
THEN
  THIS^.stSeqCtrlGeneral.strExtraInfo := 'Bitte quittieren und erneut testen';
  IF TRUE
  //AND itfOpMode.P_QUIT
  THEN
    THIS^.stSeqCtrlGeneral.eActiveSeqState := E_SEQ_GENERAL.EXECUTE;
	END_IF
  
END_IF

ELSE
  THIS^.stSeqCtrlGeneral.eActiveSeqState := E_SEQ_GENERAL.ERROR;
END_CASE
END_METHOD

METHOD PRIVATE _m_Seq_TABLE_EXIST_CHECK : E_SEQ_PROCESS
VAR_INPUT
END_VAR
VAR
	ActiveSeq: STRING;
END_VAR
//THIS^._m_GeneralStepSetting(StepType:=E_STEP_STATE_TYPE.INIT,
ActiveSeq := TO_STRING(THIS^.eSeq);

CASE THIS^.stSeqCtrlGeneral.eActiveSeqState OF
E_SEQ_GENERAL.READY:;
	
E_SEQ_GENERAL.EXECUTE:;
	IF TRUE
	THEN
		THIS^.stSeqCtrlGeneral.eActiveSeqState := E_SEQ_GENERAL.RESET;
	END_IF
  
E_SEQ_GENERAL.RESET:;
	stSeqCtrlGeneral.iInternalSeqStateCase := 0;
	IF TRUE
	THEN
		THIS^.stSeqCtrlGeneral.eActiveSeqState := E_SEQ_GENERAL.BUSY;
	END_IF
  
E_SEQ_GENERAL.BUSY:;
	CASE THIS^.stSeqCtrlGeneral.iInternalSeqStateCase OF
    0:  // Connect to database
      IF TRUE 
      AND NOT THIS^.fbSQLDatabase.bConnected
			THEN 
        IF THIS^.fbSQLDatabase.Connect(THIS^.udiDBID) THEN
          IF THIS^.fbSQLDatabase.bError THEN
            THIS^.stSeqCtrlGeneral.eActiveSeqState := E_SEQ_GENERAL.ERROR;
          ELSE
            THIS^.stSeqCtrlGeneral.iInternalSeqStateCase := 10;
          END_IF
        END_IF
      ELSE
        THIS^.stSeqCtrlGeneral.iInternalSeqStateCase := 10;
			END_IF

    10:	// Execute command
      IF TRUE 
			THEN 
        IF THIS^.fbSQLCommand.Execute(ADR(THIS^.sCmd), SIZEOF(THIS^.sCmd)) THEN
          THIS^.bResult := NOT THIS^.fbPLCDBWriteEvt.bError;
          THIS^.stSeqCtrlGeneral.iInternalSeqStateCase := 20;
        END_IF
			END_IF
      
    1220:	// Execute command
      IF TRUE
      AND fbPLCDBCmd.Execute(hDBID:= THIS^.udiDBID, 
                              pExpression:= pExpression, 
                              cbExpression:= cbExpression, 
                              pData:= pData, 
                              cbData:= cbData, 
                              pParameter:= pParameter, 
                              cbParameter:= cbParameter) 
      THEN
        THIS^.bResult := NOT THIS^.fbPLCDBWriteEvt.bError;
        THIS^.stSeqCtrlGeneral.iInternalSeqStateCase := 20;
      END_IF
      
    20:	// Disconnect
      IF TRUE 
			THEN 
        IF THIS^.fbSQLDatabase.Disconnect() THEN
          IF THIS^.fbSqlDatabase.bError THEN
            THIS^.stSeqCtrlGeneral.eActiveSeqState := E_SEQ_GENERAL.ERROR;
          ELSE
            THIS^.stSeqCtrlGeneral.iInternalSeqStateCase := 1000;
          END_IF
        END_IF
			END_IF
      
    1000: // Exit step
      IF TRUE
      THEN
        THIS^.stSeqCtrlGeneral.iInternalSeqStateCase := 9999;
			END_IF
      
	ELSE
		THIS^.stSeqCtrlGeneral.eActiveSeqState := E_SEQ_GENERAL.DONE;  
	END_CASE
	THIS^.stSeqCtrlGeneral.strExtraInfo := CONCAT('Internal state: ', TO_STRING(THIS^.stSeqCtrlGeneral.iInternalSeqStateCase));

E_SEQ_GENERAL.DONE:;

E_SEQ_GENERAL.ERROR:;

E_SEQ_GENERAL.TIME_OUT:; 

ELSE
  THIS^.stSeqCtrlGeneral.eActiveSeqState := E_SEQ_GENERAL.ERROR;
END_CASE
END_METHOD

METHOD PRIVATE _m_Seq_WRITE : E_SEQ_PROCESS
VAR_INPUT
END_VAR
VAR
	ActiveSeq: STRING;
END_VAR
//THIS^._m_GeneralStepSetting(StepType:=E_STEP_STATE_TYPE.INIT,
ActiveSeq := TO_STRING(THIS^.eSeq);

CASE THIS^.stSeqCtrlGeneral.eActiveSeqState OF
E_SEQ_GENERAL.READY:;

	
E_SEQ_GENERAL.EXECUTE:;
	IF TRUE
	THEN
		THIS^.stSeqCtrlGeneral.eActiveSeqState := E_SEQ_GENERAL.RESET;
	END_IF
  
E_SEQ_GENERAL.RESET:;
	stSeqCtrlGeneral.iInternalSeqStateCase := 0;
	IF TRUE
	THEN
		THIS^.stSeqCtrlGeneral.eActiveSeqState := E_SEQ_GENERAL.BUSY;
	END_IF
  
E_SEQ_GENERAL.BUSY:;
	CASE THIS^.stSeqCtrlGeneral.iInternalSeqStateCase OF
		0:	// Entrance step --> Create command
      IF TRUE 
			THEN 
        IF fbPLCDBWriteEvt.Write(
          hDBID:= THIS^.udiDBID, 
          sTableName:= THIS^.sTableName,
          pValue:= THIS^.pValue, 
          cbValue:= THIS^.cbValue, 
          sDBSymbolName:= THIS^.sDBSymbolName, 
          eDBWriteMode:= THIS^.eDBWriteMode, 
          nRingBuffParameter:= THIS^.nRingBuffParameter) 
        THEN
          IF fbPLCDBWriteEvt.bError THEN
            THIS^.stSeqCtrlGeneral.eActiveSeqState := E_SEQ_GENERAL.ERROR; 
          ELSE
            THIS^.stSeqCtrlGeneral.iInternalSeqStateCase := 1000;
          END_IF
        END_IF
			END_IF
      
	ELSE
		THIS^.stSeqCtrlGeneral.eActiveSeqState := E_SEQ_GENERAL.DONE;  
	END_CASE
	THIS^.stSeqCtrlGeneral.strExtraInfo := CONCAT('Internal state: ', TO_STRING(THIS^.stSeqCtrlGeneral.iInternalSeqStateCase));

E_SEQ_GENERAL.DONE:;

E_SEQ_GENERAL.ERROR:;

E_SEQ_GENERAL.TIME_OUT:; 
IF TRUE
AND THIS^.stSeqCtrlGeneral.bTimeOutActiveQuit 
THEN
  THIS^.stSeqCtrlGeneral.strExtraInfo := 'Bitte quittieren und erneut testen';
  IF TRUE
  //AND itfOpMode.P_QUIT
  THEN
    THIS^.stSeqCtrlGeneral.eActiveSeqState := E_SEQ_GENERAL.EXECUTE;
	END_IF
  
END_IF

ELSE
  THIS^.stSeqCtrlGeneral.eActiveSeqState := E_SEQ_GENERAL.ERROR;
END_CASE
END_METHOD

METHOD PRIVATE _m_Seq_WRITE_BY_SYMBOL : E_SEQ_PROCESS
VAR_INPUT
END_VAR
VAR
	ActiveSeq: STRING;
END_VAR
//THIS^._m_GeneralStepSetting(StepType:=E_STEP_STATE_TYPE.INIT,
ActiveSeq := TO_STRING(THIS^.eSeq);

CASE THIS^.stSeqCtrlGeneral.eActiveSeqState OF
E_SEQ_GENERAL.READY:;

	
E_SEQ_GENERAL.EXECUTE:;
	IF TRUE
	THEN
		THIS^.stSeqCtrlGeneral.eActiveSeqState := E_SEQ_GENERAL.RESET;
	END_IF
  
E_SEQ_GENERAL.RESET:;
	stSeqCtrlGeneral.iInternalSeqStateCase := 0;
	IF TRUE
	THEN
		THIS^.stSeqCtrlGeneral.eActiveSeqState := E_SEQ_GENERAL.BUSY;
	END_IF
  
E_SEQ_GENERAL.BUSY:;
	CASE THIS^.stSeqCtrlGeneral.iInternalSeqStateCase OF
		0:	// Entrance step --> Create command
      IF TRUE 
			THEN 
        IF fbPLCDBWriteEvt.WriteBySymbol(
          hDBID:= THIS^.udiDBID, 
          sTableName:= THIS^.sTableName, 
          stADSDevice:= THIS^.stADSDevice, 
          stSymbol:= THIS^.stSymbol, 
          eDBWriteMode:= THIS^.eDBWriteMode, 
          nRingBuffParameter:= THIS^.nRingBuffParameter) 
        THEN
          IF fbPLCDBWriteEvt.bError THEN
            THIS^.stSeqCtrlGeneral.eActiveSeqState := E_SEQ_GENERAL.ERROR; 
          ELSE
            THIS^.stSeqCtrlGeneral.iInternalSeqStateCase := 1000;
          END_IF
        END_IF
			END_IF
      
	ELSE
		THIS^.stSeqCtrlGeneral.eActiveSeqState := E_SEQ_GENERAL.DONE;  
	END_CASE
	THIS^.stSeqCtrlGeneral.strExtraInfo := CONCAT('Internal state: ', TO_STRING(THIS^.stSeqCtrlGeneral.iInternalSeqStateCase));

E_SEQ_GENERAL.DONE:;

E_SEQ_GENERAL.ERROR:;

E_SEQ_GENERAL.TIME_OUT:; 
IF TRUE
AND THIS^.stSeqCtrlGeneral.bTimeOutActiveQuit 
THEN
  THIS^.stSeqCtrlGeneral.strExtraInfo := 'Bitte quittieren und erneut testen';
  IF TRUE
  //AND itfOpMode.P_QUIT
  THEN
    THIS^.stSeqCtrlGeneral.eActiveSeqState := E_SEQ_GENERAL.EXECUTE;
	END_IF
  
END_IF

ELSE
  THIS^.stSeqCtrlGeneral.eActiveSeqState := E_SEQ_GENERAL.ERROR;
END_CASE
END_METHOD

METHOD PRIVATE _m_Seq_WRITE_STRUCT : E_SEQ_PROCESS
VAR_INPUT
END_VAR
VAR
	ActiveSeq: STRING;
END_VAR
//THIS^._m_GeneralStepSetting(StepType:=E_STEP_STATE_TYPE.INIT,
ActiveSeq := TO_STRING(THIS^.eSeq);

CASE THIS^.stSeqCtrlGeneral.eActiveSeqState OF
E_SEQ_GENERAL.READY:;

	
E_SEQ_GENERAL.EXECUTE:;
	IF TRUE
	THEN
		THIS^.stSeqCtrlGeneral.eActiveSeqState := E_SEQ_GENERAL.RESET;
	END_IF
  
E_SEQ_GENERAL.RESET:;
	stSeqCtrlGeneral.iInternalSeqStateCase := 0;
	IF TRUE
	THEN
		THIS^.stSeqCtrlGeneral.eActiveSeqState := E_SEQ_GENERAL.BUSY;
	END_IF
  
E_SEQ_GENERAL.BUSY:;
	CASE THIS^.stSeqCtrlGeneral.iInternalSeqStateCase OF
		0:	// Entrance step --> Create command
      IF TRUE 
			THEN 
        IF fbPLCDBWriteEvt.WriteStruct(hDBID:= THIS^.udiDBID, 
                                       sTableName:= THIS^.sTableName, 
                                       pRecord:= THIS^.pRecord, 
                                       cbRecord:= THIS^.cbRecord, 
                                       pColumnNames:= THIS^.pColumnNames, 
                                       cbColumnNames:= THIS^.cbColumnNames)
        THEN
          IF fbPLCDBWriteEvt.bError THEN
            THIS^.stSeqCtrlGeneral.eActiveSeqState := E_SEQ_GENERAL.ERROR; 
          ELSE
            THIS^.stSeqCtrlGeneral.iInternalSeqStateCase := 1000;
          END_IF
        END_IF
			END_IF
      
	ELSE
		THIS^.stSeqCtrlGeneral.eActiveSeqState := E_SEQ_GENERAL.DONE;  
	END_CASE
	THIS^.stSeqCtrlGeneral.strExtraInfo := CONCAT('Internal state: ', TO_STRING(THIS^.stSeqCtrlGeneral.iInternalSeqStateCase));

E_SEQ_GENERAL.DONE:;

E_SEQ_GENERAL.ERROR:;

E_SEQ_GENERAL.TIME_OUT:; 
IF TRUE
AND THIS^.stSeqCtrlGeneral.bTimeOutActiveQuit 
THEN
  THIS^.stSeqCtrlGeneral.strExtraInfo := 'Bitte quittieren und erneut testen';
  IF TRUE
  //AND itfOpMode.P_QUIT
  THEN
    THIS^.stSeqCtrlGeneral.eActiveSeqState := E_SEQ_GENERAL.EXECUTE;
	END_IF
  
END_IF

ELSE
  THIS^.stSeqCtrlGeneral.eActiveSeqState := E_SEQ_GENERAL.ERROR;
END_CASE
END_METHOD

METHOD PRIVATE _m_SequenceManager
VAR_INPUT
END_VAR
IF FALSE
//AND THIS^.eActiveSeqState=DONE 
AND eLastSeq<>eSeq
THEN
	IF THIS^.stSeqCtrlGeneral.eActiveSeqState<>E_SEQ_GENERAL.EXECUTE THEN
		THIS^.stSeqCtrlGeneral.eActiveSeqState:=E_SEQ_GENERAL.READY;
	END_IF
END_IF

eSeq := eNextSeq;

//DelayTimer und TimeOut Timer verwalten
stSeqCtrlGeneral.bActiveStep:=	TRUE
				AND eLastSeq					=	eSeq
				AND stSeqCtrlGeneral.eLastActiveSeqState			=	stSeqCtrlGeneral.eActiveSeqState
				AND	stSeqCtrlGeneral.iLastInternalSeqStateCase	=	stSeqCtrlGeneral.iInternalSeqStateCase
				;
			
IF NOT stSeqCtrlGeneral.bActiveStep THEN
	stSeqCtrlGeneral.bDelayActive:=FALSE;
	stSeqCtrlGeneral.bTimeOutActiveQuit:=FALSE;
	stSeqCtrlGeneral.bTimeOutActiveNoQuit:=FALSE;
  THIS^.stSeqCtrlGeneral.strExtraInfo:='';
END_IF

_m_SaveLastStep();
stSeqCtrlGeneral.tonDelay	(IN:=stSeqCtrlGeneral.bActiveStep AND stSeqCtrlGeneral.bDelayActive, 		PT:=stSeqCtrlGeneral.tDelay);
stSeqCtrlGeneral.tonTimeOut	(IN:=stSeqCtrlGeneral.bActiveStep AND (stSeqCtrlGeneral.bTimeOutActiveNoQuit OR stSeqCtrlGeneral.bTimeOutActiveQuit), 	PT:=stSeqCtrlGeneral.tTimeOut);
stSeqCtrlGeneral.tonStepTime	(IN:= stSeqCtrlGeneral.bActiveStep, PT:= T#24H);

IF stSeqCtrlGeneral.tonTimeOut.Q  THEN
	stSeqCtrlGeneral.eActiveSeqState:=E_SEQ_GENERAL.TIME_OUT;
END_IF

IF stSeqCtrlGeneral.iError<>0 THEN
	eSeq:=E_SEQ_DATABASE.ERROR_SEQ;
END_IF



eLastSeq					:=	eSeq;
stSeqCtrlGeneral.eLastActiveSeqState			:=	stSeqCtrlGeneral.eActiveSeqState;
stSeqCtrlGeneral.iLastInternalSeqStateCase	:=	stSeqCtrlGeneral.iInternalSeqStateCase;

// Reset set ready state
IF THIS^.stSeqCtrlGeneral.bExitSetReadyState THEN
  THIS^.stSeqCtrlGeneral.bExitSetReadyState := FALSE;
END_IF
END_METHOD

METHOD PRIVATE _m_TimeOut : BOOL
VAR_INPUT
	bTimeoutActiveToQuit:	BOOL;
	bTimeOutActiveNoQuit:	BOOL;
	tTimeOut:				TIME;	
END_VAR
THIS^.stSeqCtrlGeneral.bTimeOutActiveQuit:=	bTimeoutActiveToQuit;
THIS^.stSeqCtrlGeneral.bTimeOutActiveNoQuit:=	bTimeOutActiveNoQuit;
THIS^.stSeqCtrlGeneral.tTimeOut:=			tTimeOut;
_m_TimeOut:=FALSE;
IF THIS^.stSeqCtrlGeneral.tonTimeOut.Q THEN
	_m_TimeOut:=TRUE;
END_IF
END_METHOD

METHOD FB_init : BOOL
VAR_INPUT
	bInitRetains : BOOL; // if TRUE, the retain variables are initialized (warm start / cold start)
	bInCopyCode : BOOL;  // if TRUE, the instance afterwards gets moved into the copy code (online change)
  
  itfLogEvents: 										                      I_HANDLE_EVENTS;
  itfOpMode:											                        I_OP_MODE;  
END_VAR
THIS^.itfLogEvents := itfLogEvents;
THIS^.itfOpMode := itfOpMode;
END_METHOD

METHOD M_ClearTable : BOOL
VAR_INPUT
  /// Indicates the ID of the database to be used.
  udiDBID:          UDINT;
  /// Name of the table to be created.
  sTableName:       T_MaxString;
END_VAR
M_ClearTable := THIS^.stSeqCtrlGeneral.eActiveSeqState = E_SEQ_GENERAL.DONE;

// Assign input
THIS^.udiDBID := udiDBID;
THIS^.sTableName := sTableName;

// General
IF THIS^.stSeqCtrlGeneral.eActiveSeqState = E_SEQ_GENERAL.READY THEN
  THIS^.eNextSeq := E_SEQ_DATABASE.CLEAR_TABLE;
  THIS^.stSeqCtrlGeneral.eActiveSeqState := E_SEQ_GENERAL.EXECUTE;
END_IF
END_METHOD

METHOD M_Connect : BOOL
VAR_INPUT
  /// Indicates the ID of the database to be used.
  udiDBID:                  UDINT;
END_VAR
M_Connect := THIS^.stSeqCtrlGeneral.eActiveSeqState = E_SEQ_GENERAL.DONE;

// Assign input
THIS^.udiDBID := udiDBID;

// General
IF THIS^.stSeqCtrlGeneral.eActiveSeqState = E_SEQ_GENERAL.READY THEN
  THIS^.eNextSeq := E_SEQ_DATABASE.CONNECT;
  THIS^.stSeqCtrlGeneral.eActiveSeqState := E_SEQ_GENERAL.EXECUTE;
END_IF
END_METHOD

METHOD M_CreateDatabase : BOOL
VAR_INPUT
  /// Address of the database configuration structure
  pDatabaseConfig:  POINTER TO BYTE;
  /// Length of the database configuration structure
  cbDatabaseConfig: UDINT;
  /// Indicates whether the newly created database should be entered as new configuration entry in the XML file.
  bCreateXMLConfig: BOOL;
  /// Returns the hDBID if/when a new configuration entry was created.
  pDBID:            POINTER TO UDINT;
END_VAR
M_CreateDatabase := THIS^.stSeqCtrlGeneral.eActiveSeqState = E_SEQ_GENERAL.DONE;

// Assign input
THIS^.pDatabaseConfig :=  pDatabaseConfig;
THIS^.cbDatabaseConfig := cbDatabaseConfig;
THIS^.bCreateXMLConfig := bCreateXMLConfig;
THIS^.pDBID :=            pDBID;

// General
IF THIS^.stSeqCtrlGeneral.eActiveSeqState = E_SEQ_GENERAL.READY THEN
  THIS^.eNextSeq := E_SEQ_DATABASE.CREATE_DATABASE;
  THIS^.stSeqCtrlGeneral.eActiveSeqState := E_SEQ_GENERAL.EXECUTE;
END_IF

// Example
(*
VAR
    fbPLCDBCreate : FB_PLCDBCreateEvt(sNetID := '', tTimeout := T#5S);
    stConfigDB    : T_DBConfig_MsCompactSQL;
    hDBID         : UDINT;
    tcMessage     : I_TcMessage;
END_VAR

------------------------------------------------------------------------

stConfigDB.bAuthentification := FALSE;
stConfigDB.sServer := 'C:\Test.sdf';

IF fbPLCDBCreate.Database(
    pDatabaseConfig:= ADR(stConfigDB),
    cbDatabaseConfig := SIZEOF(stConfigDB),
    bCreateXMLConfig := TRUE,
    pDBID := ADR(hDBID))
THEN
    IF fbPLCDBCreate.bError THEN
        tcMessage := fbPLCDBCreate.ipTcResult;
        nState := 255;
    ELSE
        nState := 0;
    END_IF
END_IF
*)
END_METHOD

METHOD M_CreateTable : BOOL
VAR_INPUT
  /// Indicates the ID of the database to be used.
  udiDBID:                    UDINT;
  /// Name of the table that is to be read.
  sTableName:                 T_MaxString;
  /// Indicates the pointer address of the table structure array. The individual columns are written in this array.
  pTableCfg:                  POINTER TO ARRAY[0..MAX_DBCOLUMNS] OF ST_ColumnInfo;
  /// Indicates the length of the array in which the columns are configured.
  cbTableCfg:                 UDINT;
END_VAR
M_CreateTable := THIS^.stSeqCtrlGeneral.eActiveSeqState = E_SEQ_GENERAL.DONE;

// Assign input
THIS^.udiDBID :=    udiDBID;
THIS^.sTableName := sTableName;
THIS^.pTableCfg :=  pTableCfg;
THIS^.cbTableCfg := cbTableCfg;

// General
IF THIS^.stSeqCtrlGeneral.eActiveSeqState = E_SEQ_GENERAL.READY THEN
  THIS^.eNextSeq := E_SEQ_DATABASE.CREATE_TABLE;
  THIS^.stSeqCtrlGeneral.eActiveSeqState := E_SEQ_GENERAL.EXECUTE;
END_IF
END_METHOD

METHOD M_DeleteTable : BOOL
VAR_INPUT
  /// Indicates the ID of the database to be used.
  udiDBID:          UDINT;
  /// Name of the table that is to be read.
  sTableName:       T_MaxString;
END_VAR
M_DeleteTable := THIS^.stSeqCtrlGeneral.eActiveSeqState = E_SEQ_GENERAL.DONE;

// Assign input
THIS^.udiDBID := udiDBID;
THIS^.sTableName := sTableName;

// General
IF THIS^.stSeqCtrlGeneral.eActiveSeqState = E_SEQ_GENERAL.READY THEN
  THIS^.eNextSeq := E_SEQ_DATABASE.DELETE_TABLE;
  THIS^.stSeqCtrlGeneral.eActiveSeqState := E_SEQ_GENERAL.EXECUTE;
END_IF
END_METHOD

METHOD M_Disconnect : BOOL
M_Disconnect := THIS^.stSeqCtrlGeneral.eActiveSeqState = E_SEQ_GENERAL.DONE;

// General
IF THIS^.stSeqCtrlGeneral.eActiveSeqState = E_SEQ_GENERAL.READY THEN
  THIS^.eNextSeq := E_SEQ_DATABASE.DISCONNECT;
  THIS^.stSeqCtrlGeneral.eActiveSeqState := E_SEQ_GENERAL.EXECUTE;
END_IF
END_METHOD

METHOD M_ExecuteCmd : BOOL

VAR_INPUT
  /// Indicates the ID of the database to be used.
  udiDBID:      UDINT;
  /// Addres of the command
  pExpression:  POINTER TO BYTE;
  /// Indicates the number of command.
  cbExpression: UDINT;
  /// Address of the structure array into which the records are to be written.
  pData:        POINTER TO BYTE;
  /// Indicates the size of the structure array in bytes.
  cbData:       UDINT;
  /// Address of the structure array.
  pParameter:   POINTER TO ARRAY[0..MAX_DBCOLUMNS] OF ST_ExpParameter;
  /// Indicates the size of the parameter.
  cbParameter:  UDINT; 
END_VAR
M_ExecuteCmd := THIS^.stSeqCtrlGeneral.eActiveSeqState = E_SEQ_GENERAL.DONE;

// Assign input
THIS^.udiDBID := udiDBID;
THIS^.pExpression := pExpression;
THIS^.cbExpression := cbExpression;
THIS^.pData := pData;
THIS^.cbData := cbData;
THIS^.pParameter := pParameter;
THIS^.cbParameter := cbParameter;

// General
IF THIS^.stSeqCtrlGeneral.eActiveSeqState = E_SEQ_GENERAL.READY THEN
  THIS^.eNextSeq := E_SEQ_DATABASE.EXECUTE_CMD;
  THIS^.stSeqCtrlGeneral.eActiveSeqState := E_SEQ_GENERAL.EXECUTE;
END_IF

// Example
(*
VAR
    fbPLCDBCmd    : FB_PLCDBCmdEvt(sNetID := '', tTimeout := T#5S);
    sCmd          : STRING (1000); 
    myStruct      : ST_DataAll;
    aPara         : ARRAY[0..14] OF ST_ExpParameter;
    tcMessage     : I_TcMessage;
END_VAR

------------------------------------------------------------------------

TYPE ST_DataAll :
STRUCT
    colBigInt: LINT;
    colInteger: DINT;
    colSmallInt: INT;
    colTinyInt: BYTE;
    colBit: BOOL;
    colMoney: LREAL;
    colFloat: LREAL;
    colReal: REAL;
    colDateTime: DT;
    colNText: STRING(255);
    colNChar: STRING(10);
    colImage: ARRAY[0..255] OF BYTE;
    colNVarChar: STRING(50);
    colBinary: ARRAY[0..29] OF BYTE;
    colVarBinary: ARRAY[0..19] OF BYTE;
END_STRUCT
END_TYPE

------------------------------------------------------------------------

// set Parameter configuration
aPara[0].sParaName := 'colBigInt';    aPara[0].eParaType := E_ExpParameterType.Int64;      aPara[0].nParaSize := 8;
aPara[1].sParaName := 'colInteger';   aPara[1].eParaType := E_ExpParameterType.Int32;      aPara[1].nParaSize := 4;
aPara[2].sParaName := 'colSmallInt';  aPara[2].eParaType := E_ExpParameterType.Int16;      aPara[2].nParaSize := 2;
aPara[3].sParaName := 'colTinyInt';   aPara[3].eParaType := E_ExpParameterType.Byte_;      aPara[3].nParaSize := 1;
aPara[4].sParaName := 'colBit';       aPara[4].eParaType := E_ExpParameterType.Boolean;    aPara[4].nParaSize := 1;
aPara[5].sParaName := 'colMoney';     aPara[5].eParaType := E_ExpParameterType.Double64;   aPara[5].nParaSize := 8;
aPara[6].sParaName := 'colFloat';     aPara[6].eParaType := E_ExpParameterType.Double64;   aPara[6].nParaSize := 8;
aPara[7].sParaName := 'colReal';      aPara[7].eParaType := E_ExpParameterType.Float32;    aPara[7].nParaSize := 4;
aPara[8].sParaName := 'colDateTime';  aPara[8].eParaType := E_ExpParameterType.DateTime;   aPara[8].nParaSize := 4;
aPara[9].sParaName := 'colNText';     aPara[9].eParaType := E_ExpParameterType.STRING_;    aPara[9].nParaSize := 256;
aPara[10].sParaName:= 'colNChar';     aPara[10].eParaType := E_ExpParameterType.STRING_;   aPara[10].nParaSize := 10;
aPara[11].sParaName:= 'colImage';     aPara[11].eParaType := E_ExpParameterType.ByteArray; aPara[11].nParaSize := 256;
aPara[12].sParaName:= 'colNVarChar';  aPara[12].eParaType := E_ExpParameterType.STRING_;   aPara[12].nParaSize := 50;
aPara[13].sParaName:= 'colBinary';    aPara[13].eParaType := E_ExpParameterType.ByteArray; aPara[13].nParaSize := 30;
aPara[14].sParaName:= 'colVarBinary'; aPara[14].eParaType := E_ExpParameterType.ByteArray; aPara[14].nParaSize := 20;

// set command
sCmd := 'INSERT INTO MyTableName (colInteger, colSmallInt, colTinyInt, colBit, colMoney, colFloat, colReal, colDateTime, colNText, colNChar, colImage, colNVarChar, colBinary, colVarBinary) VALUES ({colInteger}, {colSmallInt}, {colTinyInt}, {colBit}, {colMoney}, {colFloat}, {colReal}, {colDateTime}, {colNText}, {colNChar}, {colImage}, {colNVarChar}, {colBinary}, {colVarBinary})';

// call functionblock
IF fbPLCDBCmd.Execute(
    hDBID:= 1, 
    pExpression:= ADR(sCmd), 
    cbExpression:= SIZEOF(sCmd), 
    pData:= ADR(myStruct), 
    cbData:= SIZEOF(myStruct), 
    pParameter:= ADR(aPara), 
    cbParameter:= SIZEOF(aPara)) 
THEN
    IF fbPLCDBCmd.bError THEN
        tcMessage := fbPLCDBCmd.ipTcResult;
        nState := 255; 
    ELSE
        nState := 0;
    END_IF
END_IF
*)
END_METHOD

METHOD M_ExecuteSimplifyCmd : BOOL

VAR_INPUT
  /// Indicates the ID of the database to be used.
  udiDBID:      UDINT;
  /// Indicates the pointer address of a string variable with the SQL command to be executed.
  pSQLCmd:      POINTER TO BYTE;
  /// Indicates the length of a SQL command to be executed.
  cbSQLCmd:     UDINT;
END_VAR
M_ExecuteSimplifyCmd := THIS^.stSeqCtrlGeneral.eActiveSeqState = E_SEQ_GENERAL.DONE;

// Assign input
THIS^.udiDBID := udiDBID;
THIS^.pSQLCmd := pSQLCmd;
THIS^.cbSQLCmd := cbSQLCmd;

// General
IF THIS^.stSeqCtrlGeneral.eActiveSeqState = E_SEQ_GENERAL.READY THEN
  THIS^.eNextSeq := E_SEQ_DATABASE.EXECUTE_SIMPLIFY_CMD;
  THIS^.stSeqCtrlGeneral.eActiveSeqState := E_SEQ_GENERAL.EXECUTE;
END_IF

// Example
(*
VAR
    fbSqlCommand : FB_SQLCommandEvt(sNetID := '', tTimeout := T#5S);
    tcMessage    : I_TcMessage;
END_VAR

------------------------------------------------------------------------

// you can generate this with the SQL Query Editor 
sCmd := 'INSERT INTO myTable_Double ( Timestamp, Name, Value) VALUES ( $'2018-01-31 14:59:27$', $'Temperature$', 21.3)';

// call sql command
IF fbSQLCommand.Execute(ADR(sCmd), SIZEOF(sCmd)) THEN
    IF fbSQLCommand.bError THEN
        tcMessage := fbSQLCommand.ipTcResult;
        nState := 255; 
    ELSE
        nState := nState+1; 
    END_IF
END_IF
*)
END_METHOD

METHOD M_Overwrite : BOOL

VAR_INPUT
  /// Indicates the ID of the database to be used.
  udiDBID:                    UDINT;
  /// Name of the table that is to be read.
  sTableName:                 T_MaxString;
  /// Column name of the data to be updated
  sColumnNameToUpdate:        STRING;
  /// Column value of the data to be updated
  sColumnValToUpdate:         STRING;
  /// Column name to set
  sColumnNameToSet:           STRING;
  /// New value
  sNewVal:                    STRING;
END_VAR
M_Overwrite := THIS^.stSeqCtrlGeneral.eActiveSeqState = E_SEQ_GENERAL.DONE;

// Assign input
THIS^.udiDBID := udiDBID;
THIS^.sTableName := sTableName;
THIS^.sColumnNameToUpdate := sColumnNameToUpdate;
THIS^.sColumnValToUpdate := sColumnValToUpdate;
THIS^.sColumnNameToSet := sColumnNameToSet;
THIS^.sNewVal := sNewVal;

// General
IF THIS^.stSeqCtrlGeneral.eActiveSeqState = E_SEQ_GENERAL.READY THEN
  THIS^.eNextSeq := E_SEQ_DATABASE.OVERWRITE;
  THIS^.stSeqCtrlGeneral.eActiveSeqState := E_SEQ_GENERAL.EXECUTE;
END_IF
END_METHOD

METHOD M_Read : BOOL

VAR_INPUT
  /// Indicates the ID of the database to be used.
  udiDBID:                    UDINT;
  /// Name of the table that is to be read.
  sTableName:                 T_MaxString;
  /// Symbol name to be read from the standard table structure.
  sDBSymbolName:              STRING;
  /// Sorting column (ID, timestamp, name or value)
  eOrderBy:                   E_OrderColumn;
  /// Sorting direction (ASC or DESC)
  eOrderType:                 E_OrderType;
  /// Indicates the index of the first record to be read.
  nStartIndex:                UDINT;
  /// Indicates the number of records to be read.
  nRecordCount:               UDINT;
  /// Address of the structure array into which the records are to be written.
  pData2:                     POINTER TO ST_StandardRecord;
  /// Indicates the size of the structure array in bytes.
  cbData:                     UDINT;
END_VAR
VAR
  
END_VAR
M_Read := THIS^.stSeqCtrlGeneral.eActiveSeqState = E_SEQ_GENERAL.DONE;

// Assign input
THIS^.udiDBID := udiDBID;
THIS^.sTableName := sTableName;
THIS^.sDBSymbolName := sDBSymbolName;
THIS^.eOrderBy := eOrderBy;
THIS^.eOrderType := eOrderType;
THIS^.nStartIndex := nStartIndex;
THIS^.nRecordCount := nRecordCount;
THIS^.pData2 := pData2;
THIS^.cbData := cbData;

// General
IF THIS^.stSeqCtrlGeneral.eActiveSeqState = E_SEQ_GENERAL.READY THEN
  THIS^.eNextSeq := E_SEQ_DATABASE.READ;
  THIS^.stSeqCtrlGeneral.eActiveSeqState := E_SEQ_GENERAL.EXECUTE;
END_IF

// Example
(*
VAR
    fbPLCDBRead    : FB_PLCDBReadEvt (sNetID := '', tTimeout := T#5S);
    ReadStruct     : ST_StandardRecord;
    tcMessage      : I_TcMessage;
END_VAR

------------------------------------------------------------------------

IF fbPLCDBRead.Read(
    hDBID:= 1, 
    sTableName:= 'MyTable_WithLReal', 
    sDBSymbolName:= 'MyValue', 
    eOrderBy:= E_OrderColumn.ID, 
    eOrderType:= E_OrderType.DESC, 
    nStartIndex:= 0, 
    nRecordCount:= 1, 
    pData:= ADR(ReadStruct), 
    cbData:= SIZEOF(ReadStruct))
THEN
    IF fbPLCDBRead.bError THEN
        tcMessage := fbPLCDBRead.ipTcResult;
        nState := 255; 
    ELSE
        nState := 0;
    END_IF
END_IF
*)
END_METHOD

METHOD M_ReadStruct : BOOL

VAR_INPUT
  /// Indicates the ID of the database to be used.
  udiDBID:                    UDINT;
  /// Name of the table that is to be read.
  sTableName:                 T_MaxString;
  /// Address of the array containing the column name to be read.
  pColumnNames:               POINTER TO ARRAY [0..MAX_DBCOLUMNS] OF STRING(50);
  /// Length of the column name array
  cbColumnNames:              UDINT;
  /// Name the sorting column
  sOrderByColumn:             STRING(50);
  /// Sorting direction (ASC or DESC)
  eOrderType:                 E_OrderType;
  /// Indicates the index of the first record to be read.
  nStartIndex:                UDINT;
  /// Indicates the number of records to be read.
  nRecordCount:               UDINT;
  /// Address of the structure array into which the records are to be written.
  pData:                      POINTER TO BYTE;
  /// Indicates the size of the structure array in bytes.
  cbData:                     UDINT;
END_VAR
VAR
  
END_VAR
M_ReadStruct := THIS^.stSeqCtrlGeneral.eActiveSeqState = E_SEQ_GENERAL.DONE;

// Assign input
THIS^.udiDBID := udiDBID;
THIS^.sTableName := sTableName;
THIS^.pColumnNames := pColumnNames;
THIS^.cbColumnNames := cbColumnNames;
THIS^.sOrderByColumn := sOrderByColumn;
THIS^.eOrderType := eOrderType;
THIS^.nStartIndex := nStartIndex;
THIS^.nRecordCount := nRecordCount;
THIS^.pData := pData;
THIS^.cbData := cbData;

// General
IF THIS^.stSeqCtrlGeneral.eActiveSeqState = E_SEQ_GENERAL.READY THEN
  THIS^.eNextSeq := E_SEQ_DATABASE.READ_STRUCT;
  THIS^.stSeqCtrlGeneral.eActiveSeqState := E_SEQ_GENERAL.EXECUTE;
END_IF

// Example
(*
VAR
    fbPLCDBRead    : FB_PLCDBReadEvt (sNetID := '', tTimeout := T#5S);
    myCustomStruct : ST_Record;
    tcMessage      : I_TcMessage;
END_VAR

------------------------------------------------------------------------

TYPE ST_Record :
STRUCT
    nID        : LINT;
    dtTimestamp: DATE_AND_TIME;
    sName      : STRING;
    nSensor1   : LREAL;
    nSensor2   : LREAL;
END_STRUCT
END_TYPE

--------------------------------------------------------------------------

// set columnnames
ColumnNames[0] := 'ID';
ColumnNames[1] := 'Timestamp';
ColumnNames[2] := 'Name';
ColumnNames[3] := 'Sensor1';
ColumnNames[4] := 'Sensor2';

IF fbPLCDBRead.ReadStruct(
    hDBID:= 1, 
    sTableName:= 'MyTable_Struct', 
    pColumnNames:= ADR(ColumnNames), 
    cbColumnNames:= SIZEOF(ColumnNames), 
    sOrderByColumn:= ColumnNames[0], 
    eOrderType:= E_OrderType.DESC, 
    nStartIndex:= 0, 
    nRecordCount:= 1, 
    pData:= ADR(myCustomStruct), 
    cbData:= SIZEOF(myCustomStruct))
THEN
    IF fbPLCDBRead.bError THEN
        tcMessage:= fbPLCDBRead.ipTcResult;
        nState := 255; 
    ELSE
        nState := 0;
    END_IF
END_IF
*)
END_METHOD

METHOD M_Reset : BOOL
M_Reset := THIS^.stSeqCtrlGeneral.eActiveSeqState = E_SEQ_GENERAL.DONE;

// General
IF THIS^.stSeqCtrlGeneral.eActiveSeqState = E_SEQ_GENERAL.READY THEN
  THIS^.eNextSeq := E_SEQ_DATABASE.INIT;
  THIS^.stSeqCtrlGeneral.eActiveSeqState := E_SEQ_GENERAL.EXECUTE;
END_IF
END_METHOD

(*=== Method: M_Run  ============================================

 @brief: Here is the global code (Timer, Event, Flange,...)*)
METHOD M_Run
END_METHOD

METHOD M_SetReady : BOOL
VAR_INPUT
END_VAR
M_SetReady := TRUE
              AND THIS^.stSeqCtrlGeneral.eActiveSeqState = E_SEQ_GENERAL.READY
              AND THIS^.eSeq = E_SEQ_DATABASE.BASE;

THIS^.stSeqCtrlGeneral.eActiveSeqState := E_SEQ_GENERAL.READY;
THIS^.eNextSeq := E_SEQ_DATABASE.BASE;
END_METHOD

METHOD M_TableExistCheck : BOOL
VAR_INPUT
  /// Indicates the ID of the database to be used.
  udiDBID:                    UDINT;
  /// Name of the table that is to be read.
  sTableName:                 T_MaxString;
END_VAR
VAR_OUTPUT
  /// Result
  bResult:                    BOOL;
END_VAR
M_TableExistCheck := THIS^.stSeqCtrlGeneral.eActiveSeqState = E_SEQ_GENERAL.DONE;

// Assign input
THIS^.udiDBID := udiDBID;
THIS^.sTableName := sTableName;
THIS^.sCmd := CONCAT('SELECT * FROM $'', sTableName);
THIS^.sCmd := CONCAT(THIS^.sCmd, '$'');
THIS^.pSQLCmd := ADR(THIS^.sCmd);
THIS^.cbSQLCmd := SIZEOF(THIS^.sCmd);

// Assign output
bResult := THIS^.bResult;

// General
IF THIS^.stSeqCtrlGeneral.eActiveSeqState = E_SEQ_GENERAL.READY THEN
  THIS^.eNextSeq := E_SEQ_DATABASE.TABLE_EXIST_CHECK;
  THIS^.stSeqCtrlGeneral.eActiveSeqState := E_SEQ_GENERAL.EXECUTE;
END_IF
END_METHOD

METHOD M_Write : BOOL

VAR_INPUT
  /// Indicates the ID of the database to be used.
  udiDBID:            UDINT;
  /// Name of the table that is to be write.
  sTableName:         T_MaxString;
  /// Address of the variable to be logged in the standard table structure.
  pValue:             POINTER TO BYTE;
  /// Length of the variable to be logged.
  cbValue:            UDINT;
  /// Name that is logged in the table.
  sDBSymbolName:      STRING;
  /// Indicates the write mode. (append, update, ring buffer)
  eDBWriteMode:       E_WriteMode;
  /// Additional parameter(s) for the "ring buffer" write mode.
  nRingBuffParameter: UDINT;
END_VAR
M_Write := THIS^.stSeqCtrlGeneral.eActiveSeqState = E_SEQ_GENERAL.DONE;

// Assign input
THIS^.udiDBID := udiDBID;
THIS^.sTableName := sTableName;
THIS^.pValue := pValue;
THIS^.cbValue := cbValue;
THIS^.sDBSymbolName := sDBSymbolName;
THIS^.eDBWriteMode := eDBWriteMode;
THIS^.nRingBuffParameter := nRingBuffParameter;

// General
IF THIS^.stSeqCtrlGeneral.eActiveSeqState = E_SEQ_GENERAL.READY THEN
  THIS^.eNextSeq := E_SEQ_DATABASE.WRITE;
  THIS^.stSeqCtrlGeneral.eActiveSeqState := E_SEQ_GENERAL.EXECUTE;
END_IF

// Example
(*
VAR
    fbPLCDBWrite    : FB_PLCDBWriteEvt(sNetID := '', tTimeout := T#5S);
    myValue         : LREAL := 43.23;
    tcMessage       : I_TcMessage;
END_VAR

------------------------------------------------------------------------

IF fbPLCDBWrite.Write(
    hDBID:= 1, 
    sTableName:= 'myTable_WithLReal',
    pValue:= ADR(myValue), 
    cbValue:= SIZEOF(myValue), 
    sDBSymbolName:= 'MyValue', 
    eDBWriteMode:= E_WriteMode.eADS_TO_DB_RingBuff_Count, 
    nRingBuffParameter:= 3) 
THEN
    IF fbPLCDBWrite.bError THEN
        tcMessage := fbPLCDBWrite.ipTcResult;
        nState := 255; 
    ELSE
        nState := 0; 
    END_IF
END_IF
*)
END_METHOD

METHOD M_WriteBySymbol : BOOL

VAR_INPUT
  /// Indicates the ID of the database to be used.
  udiDBID:            UDINT;
  /// Name of the table that is to be write.
  sTableName:         T_MaxString;
  /// ADS device from which a symbol is to be logged in the standard table structure.
  stADSDevice:        ST_ADSDevice;
  /// Symbol name of the variable to be written
  stSymbol:           ST_Symbol;
  /// Indicates the write mode. (append, update, ring buffer)
  eDBWriteMode:       E_WriteMode;
  /// Additional parameter(s) for the "ring buffer" write mode.
  nRingBuffParameter: UDINT;
END_VAR
M_WriteBySymbol := THIS^.stSeqCtrlGeneral.eActiveSeqState = E_SEQ_GENERAL.DONE;

// Assign input
THIS^.udiDBID := udiDBID;
THIS^.sTableName := sTableName;
THIS^.stADSDevice := stADSDevice;
THIS^.stSymbol := stSymbol;
THIS^.eDBWriteMode := eDBWriteMode;
THIS^.nRingBuffParameter := nRingBuffParameter;



// General
IF THIS^.stSeqCtrlGeneral.eActiveSeqState = E_SEQ_GENERAL.READY THEN
  THIS^.eNextSeq := E_SEQ_DATABASE.WRITE_BY_SYMBOL;
  THIS^.stSeqCtrlGeneral.eActiveSeqState := E_SEQ_GENERAL.EXECUTE;
END_IF

// Example
(*
VAR
    fbPLCDBWrite    :  FB_PLCDBWriteEvt(sNetID := '', tTimeout := T#5S);
    myValue         :  LREAL := 43.23;
    myAdsDevice     :  ST_ADSDevice;
    mySymbol        :  ST_Symbol;
    tcMessage       :  I_TcMessage;
END_VAR

------------------------------------------------------------------------

// Set ADSDevice Information
myAdsDevice.sDevNetID     := '127.0.0.1.1.1';
myAdsDevice.nDevPort      := 851;
myAdsDevice.eADSRdWrtMode := E_ADSRdWrtMode.bySymbolName; 
myAdsDevice.tTimeout      := T#5S; 

// Set Symbol Information
mySymbol.eDataType        := E_PLCDataType.eType_LREAL;
mySymbol.sDBSymbolName    := 'MySymbol';
mySymbol.sSymbolName      := 'MAIN.myValue';
mySymbol.nBitSize         := 8;

// Call Functionblock
IF fbPLCDBWrite.WriteBySymbol(
    hDBID:= 1, 
    sTableName:= 'myTable_WithLReal', 
    stADSDevice:= myAdsDevice, 
    stSymbol:= mySymbol, 
    eDBWriteMode:= E_WriteMode.eADS_TO_DB_Append, 
    nRingBuffParameter:= 1) 
THEN
    IF fbPLCDBWrite.bError THEN
        tcMessage := fbPLCDBWrite.ipTcResult;
        nState := 255; 
    ELSE
        nState := 0;
    END_IF
END_IF
*)
END_METHOD

METHOD M_WriteStruct : BOOL
VAR_INPUT
  /// Indicates the ID of the database to be used.
  udiDBID:        UDINT;
  /// Name of the table that is to be write.
  sTableName:     T_MaxString;
  /// Address of a structure that is to be logged in a freely selectable table structure.
  pRecord:        POINTER TO BYTE;
  /// Length of the structure to be written
  cbRecord:       UDINT;
  /// Address of the array containing the column name to be filled.
  pColumnNames:   POINTER TO ARRAY [0..MAX_DBCOLUMNS] OF STRING(50);
  /// Length of the column name array
  cbColumnNames:  UDINT;
END_VAR
M_WriteStruct := THIS^.stSeqCtrlGeneral.eActiveSeqState = E_SEQ_GENERAL.DONE;

// Assign input
THIS^.udiDBID := udiDBID;
THIS^.sTableName := sTableName;
THIS^.pRecord := pRecord;
THIS^.cbRecord := cbRecord;
THIS^.pColumnNames := pColumnNames;
THIS^.cbColumnNames := cbColumnNames;

// General
IF THIS^.stSeqCtrlGeneral.eActiveSeqState = E_SEQ_GENERAL.READY THEN
  THIS^.eNextSeq := E_SEQ_DATABASE.WRITE_STRUCT;
  THIS^.stSeqCtrlGeneral.eActiveSeqState := E_SEQ_GENERAL.EXECUTE;
END_IF

// Example
(*
VAR
    fbPLCDBWrite    :  FB_PLCDBWriteEvt(sNetID := '', tTimeout := T#5S);
    myRecord        :  ST_Record;
    ColumnNames     :  ARRAY[0..4] OF STRING(50);
    
    systime         :  GETSYSTEMTIME;
    currentTime     :  T_FILETIME;
    tcMessage       :  I_TcMessage;
END_VAR

------------------------------------------------------------------------

TYPE ST_Record :
STRUCT
    nID        : LINT;
    dtTimestamp: DATE_AND_TIME;
    sName      : STRING;
    nSensor1   : LREAL;
    nSensor2   : LREAL;
END_STRUCT
END_TYPE

------------------------------------------------------------------------

// set Values
systime(timeLoDw => currentTime.dwLowDateTime, timeHiDW => currentTime.dwHighDateTime );
myRecord.dtTimestamp := FILETIME_TO_DT(currentTime);
myRecord.sName       := 'MyStructVal';
myRecord.nSensor1    := 12.34;
myRecord.nSensor2    := 102.5;

// set columnnames
ColumnNames[0] := 'ID';
ColumnNames[1] := 'Timestamp';
ColumnNames[2] := 'Name';
ColumnNames[3] := 'Sensor1';
ColumnNames[4] := 'Sensor2';

// Call Functionblock
IF fbPLCDBWrite.WriteStruct(
    hDBID:= 1, 
    sTableName:= 'myTable_Struct', 
    pRecord:= ADR(myRecord), 
    cbRecord:= SIZEOF(myRecord), 
    pColumnNames:= ADR(ColumnNames) , 
    cbColumnNames:= SIZEOF(ColumnNames))
THEN
    IF fbPLCDBWrite.bError THEN
        tcMessage := fbPLCDBWrite.ipTcResult;
        nState := 255; 
    ELSE
        nState := 0;
    END_IF
END_IF
*)
END_METHOD

PROPERTY P_Connected : BOOL
GET
P_Connected := THIS^.fbSQLDatabase.bConnected;
END_GET
END_PROPERTY

{warning 'Eigenschaftenimplementierung hinzufügen'}
PROPERTY P_Error : BOOL
GET
P_Error := THIS^.stSeqCtrlGeneral.eActiveSeqState = E_SEQ_GENERAL.ERROR;
END_GET
END_PROPERTY

{warning 'Eigenschaftenimplementierung hinzufügen'}
(*=== Property: P_Event  ============================================

 @param [set]: 	Set the Structure "ST_EVENT" from another Object
 @param [get]: 	Return the Structure "ST_EVENT", it contains the actual 
					event of the Object *)
PROPERTY P_Event : GenLib.ST_EVENT
GET
END_GET
SET
END_SET
END_PROPERTY

{warning 'Eigenschaftenimplementierung hinzufügen'}
(*=== Property: P_FullObjectPath  ============================================

 @param [set]: 	Set the Object Path (Clear String of Object)
 @param [get]: 	Return the Objectpath *)
PROPERTY P_FullObjectPath : STRING
GET
P_FullObjectPath:= THIS^.strFullObjectPath;
END_GET
SET
THIS^.strFullObjectPath:=P_FullObjectPath;
END_SET
END_PROPERTY

{warning 'Eigenschaftenimplementierung hinzufügen'}
(*=== Property: P_Global_Ack  ============================================

 @param [set]: 	Set the Bit for Ack from another Object
 @param [get]: 	Return the state of Ack Bit*)
PROPERTY P_Global_Ack : BOOL
GET
END_GET
SET
END_SET
END_PROPERTY

{warning 'Eigenschaftenimplementierung hinzufügen'}
(*=== Property: P_GlobalID  ============================================

 @param [set]: 	-
 @param [get]: 	Return the string of instance path*)
PROPERTY P_GlobalID : STRING
GET
P_GlobalID:= THIS^.strInstancePath;
END_GET
END_PROPERTY

END_FUNCTION_BLOCK

(* stored: Version 1.1.0.1, ProductVersion 3.1.4024.12
   POU FB_MY_SQL: Id {a5d2bb9d-5ffb-4644-ad88-027e41b4609f}, SpecialFunc None
   Folder PRIVAT: Id {3ecc3fb9-e647-4b89-8bc9-53af2aa57afa}
   Folder SEQUENCE: Id {30e1fef3-4b35-4ebf-ac3b-7885f899d9f4}
   Method _m_DebugManager: Id {00bf47e2-3537-432d-8210-8bad1315066e}
   Method _m_Delay: Id {240876ed-3e16-475a-8291-067b56bf9e1a}
   Method _m_GeneralStepSetting: Id {982c89d8-c42d-498d-ad2c-fc16adf9e1af}
   Method _m_SaveLastStep: Id {f05d8bd2-28dc-4322-86a8-231a7e99a227}
   Method _m_Seq_CLEAR_TABLE: Id {6f10cc55-6c30-4247-ae41-d88e26d8fff1}
   Method _m_Seq_CONNECT: Id {7edb053f-e4bd-4bb5-8bb3-281e16272eb5}
   Method _m_Seq_CREATE_DATABASE: Id {6906ec39-dab7-4fa9-8541-df604145f89c}
   Method _m_Seq_CREATE_TABLE: Id {5b07000f-cefe-4e29-ab45-6a4d46dedb9e}
   Method _m_Seq_DELETE_TABLE: Id {33b10fdb-90bc-422f-97a9-8bc322f31152}
   Method _m_Seq_DISCONNECT: Id {1810e8d7-dcd6-4fba-910f-0effd481e351}
   Method _m_Seq_EXECUTE_CMD: Id {4719530e-9882-4d3d-b774-5d6c6bfc507f}
   Method _m_Seq_EXECUTE_SIMPLIFY_CMD: Id {22435480-8162-48f4-a03a-65782974972d}
   Method _m_Seq_INIT: Id {49bdb870-039c-4bb9-89ab-80b2e65aa415}
   Method _m_Seq_OVERWRITE: Id {4267e0bf-7708-46e7-b5d2-83abe524ca55}
   Method _m_Seq_READ: Id {c6eb33ee-c783-4755-bf2b-8434c136739e}
   Method _m_Seq_READ_STRUCT: Id {20754c4d-5828-4d91-92fd-fc64af3f84fb}
   Method _m_Seq_TABLE_EXIST_CHECK: Id {a57a85ff-9a35-4ab8-b56d-6fb86ae12aab}
   Method _m_Seq_WRITE: Id {26f07169-0960-40e4-a38c-382821e08b10}
   Method _m_Seq_WRITE_BY_SYMBOL: Id {a2f474d5-e815-49f1-8210-c5fe9166dfcc}
   Method _m_Seq_WRITE_STRUCT: Id {2aa13154-ffd3-4b89-aada-fc5b69e401e6}
   Method _m_SequenceManager: Id {60aa4f53-83f4-4967-b5fe-acc9348a0a98}
   Method _m_TimeOut: Id {cc963fad-f45c-4656-85c7-e5837b78b9ee}
   Method FB_init: Id {84b2682d-5fce-4ea6-a885-eb96c5320f99}
   Method M_ClearTable: Id {957197e5-c9ec-42f0-b2c4-9e1dc217ed49}
   Method M_Connect: Id {a38fb75a-3fb3-42b0-9cde-1c4a0fee5c48}
   Method M_CreateDatabase: Id {4150bdfa-b812-41dd-a4a3-d584be393774}
   Method M_CreateTable: Id {3678855a-1f60-4053-b879-83b4183fa3b6}
   Method M_DeleteTable: Id {c2ee9fbd-c43c-422d-a54b-9727a71d95c4}
   Method M_Disconnect: Id {19959a7e-df75-4581-90f9-4e5cc817e7a5}
   Method M_ExecuteCmd: Id {6f5cc6e5-c2e2-49b9-bb56-a0bcc979e2a3}
   Method M_ExecuteSimplifyCmd: Id {432763c8-3e11-458d-a428-1af57e90bbba}
   Method M_Overwrite: Id {e14e6825-92f4-4c87-a469-713b52a4d8db}
   Method M_Read: Id {ace8e153-6e0e-4830-9810-5dc0260e0d02}
   Method M_ReadStruct: Id {375daaef-b995-4eab-8994-6d31c37e4754}
   Method M_Reset: Id {18c4b1fc-4909-475d-8066-0ab005ea4ce1}
   Method M_Run: Id {f785b34d-7c81-4598-865f-3154dbdb0099}
   Method M_SetReady: Id {864cc823-ef87-406e-bd56-5eb9ac6f2506}
   Method M_TableExistCheck: Id {a25a1233-81ff-4da6-a242-f213125603ba}
   Method M_Write: Id {59c4aaaf-03ee-4f5f-997b-0e20b656ed4c}
   Method M_WriteBySymbol: Id {a2425eef-b27e-4511-8ab8-019ceefc2100}
   Method M_WriteStruct: Id {50c09ae4-e091-4d87-9206-a53f7d7ccb9b}
   Property P_Connected: Id {27eaca5b-b514-40eb-8773-8d7eb1ba9719}
   Get Get: Id {dd4ece73-3d45-4465-910c-2a8e3d408a99}
   Property P_Error: Id {4e2c052b-ca46-4905-b754-99c18b2579d6}
   Get Get: Id {4b4dc93f-7ee7-4681-bc38-64ad18a63e01}
   Property P_Event: Id {5cb8184d-18a5-4e97-ac76-e4052b661574}
   Get Get: Id {85dbc100-0827-42cd-8087-fe9072655147}
   Set Set: Id {67747551-feed-4aa3-8a55-aa51daad87d7}
   Property P_FullObjectPath: Id {c7441eea-4a32-454b-851e-528c478f2a29}
   Get Get: Id {b599a773-3439-46ee-b1f6-2d762563ac8a}
   Set Set: Id {57131e7f-7577-4a93-aa9f-eded12c6187f}
   Property P_Global_Ack: Id {e3c6e5a9-809c-4c64-80a0-f53163257cd5}
   Get Get: Id {ffa7f4e7-75e8-45fd-8457-090dc4465d2f}
   Set Set: Id {9de80ecd-6381-40ed-a73e-d57f4efc9f6d}
   Property P_GlobalID: Id {fbdcfe21-2e60-4d5f-a2f7-8419e3193f67}
   Get Get: Id {4ffb3299-ba1d-4351-999d-fc78de208825} *)
